Assert.ThatWideString(
	actual := caughtMessage,
	message := "Parse an array root"
).ToBe(expected := "Invalid JSON configuration: not an object");

_Doc := '12345';

caughtMessage := TOF_Core.WideStrings.Empty;

__TRY
	root := _Reader.Parse(document := _Doc);
__CATCH(exceptionCode)
	caughtMessage := getInvalidDocumentMessage(
		exceptionCode := exceptionCode,
		catchPointPOUName := __POUNAME(),
		catchPointPosition := __POSITION()
	);
__ENDTRY

Assert.ThatWideString(
	actual := caughtMessage,
	message := "Parse a scalar root"
).ToBe(expected := "Invalid JSON configuration: not an object");
END_METHOD

(*!
<summary>Verifies successful document open with an object root.</summary>
*)
METHOD PRIVATE testOpenObjectRoot
VAR
	root : TOF_Core.CONFIGURATION_NODE;
END_VAR
_Doc := '{"key": 123}';
root := _Reader.Parse(document := _Doc);

Assert.ThatBool(actual := _Reader.IsPresent(node := root)).IsTrue();
END_METHOD

(*!
<summary>Verifies destination validation, shape checking, type mismatch and capacity errors in ReadValue.</summary>
*)
METHOD PRIVATE testReadValueValidationAndErrors
VAR
	root : TOF_Core.CONFIGURATION_NODE;
	numNode : TOF_Core.CONFIGURATION_NODE;
	strNode : TOF_Core.CONFIGURATION_NODE;
	nullNode : TOF_Core.CONFIGURATION_NODE;
	arrNode : TOF_Core.CONFIGURATION_NODE;
	objNode : TOF_Core.CONFIGURATION_NODE;
	emptyNode : TOF_Core.CONFIGURATION_NODE;
	dstDint : DINT;
	dstStr : STRING(80);
	tinyStr : STRING(2);
END_VAR
_Doc := '{"num": 42, "str": "hello world", "nullVal": null, "arr": [1], "obj": {}}';
root := _Reader.Parse(document := _Doc);
numNode := _Reader.GetField(node := root, name := 'num');
strNode := _Reader.GetField(node := root, name := 'str');
nullNode := _Reader.GetField(node := root, name := 'nullVal');
arrNode := _Reader.GetField(node := root, name := 'arr');
objNode := _Reader.GetField(node := root, name := 'obj');

expectReadValueFailure(
	node := numNode,
	valueType := TOF_Core.CONFIGURATION_VALUE_TYPE.TYPE_DINT,
	data := 0,
	size := 4,
	message := "ReadValue with a null destination",
	expected := "Invalid JSON configuration: type/size mismatch"
);

expectReadValueFailure(
	node := numNode,
	valueType := TOF_Core.CONFIGURATION_VALUE_TYPE.TYPE_DINT,
	data := ADR(dstDint),
	size := 0,
	message := "ReadValue with zero destination size",
	expected := "Invalid JSON configuration: type/size mismatch"
);

expectReadValueFailure(
	node := emptyNode,
	valueType := TOF_Core.CONFIGURATION_VALUE_TYPE.TYPE_DINT,
	data := ADR(dstDint),
	size := 4,
	message := "ReadValue with an absent node",
	expected := "Invalid JSON configuration: missing field"
);

expectReadValueFailure(
	node := nullNode,
	valueType := TOF_Core.CONFIGURATION_VALUE_TYPE.TYPE_DINT,
	data := ADR(dstDint),
	size := 4,
	message := "ReadValue on a null value",
	expected := "Invalid JSON configuration: type/size mismatch"
);

expectReadValueFailure(
	node := arrNode,
	valueType := TOF_Core.CONFIGURATION_VALUE_TYPE.TYPE_DINT,
	data := ADR(dstDint),
	size := 4,
	message := "ReadValue on an array",
	expected := "Invalid JSON configuration: type/size mismatch"
);

expectReadValueFailure(
	node := objNode,
	valueType := TOF_Core.CONFIGURATION_VALUE_TYPE.TYPE_DINT,
	data := ADR(dstDint),
	size := 4,
	message := "ReadValue on an object",
	expected := "Invalid JSON configuration: type/size mismatch"
);

expectReadValueFailure(
	node := numNode,
	valueType := TOF_Core.CONFIGURATION_VALUE_TYPE.TYPE_DINT,
	data := ADR(dstDint),
	size := 3,
	message := "ReadValue with the wrong DINT size",
	expected := "Invalid JSON configuration: type/size mismatch"
);

// SA0175: ReadValue targets a raw string buffer; no character indexing is performed.
{analysis -175}
expectReadValueFailure(
	node := numNode,
	valueType := TOF_Core.CONFIGURATION_VALUE_TYPE.TYPE_STRING,
	data := ADR(dstStr),
	size := SIZEOF(dstStr),
	message := "ReadValue into STRING from a number",
	expected := "Invalid JSON configuration: type/size mismatch"
);

expectReadValueFailure(
	node := strNode,
	valueType := TOF_Core.CONFIGURATION_VALUE_TYPE.TYPE_STRING,
	data := ADR(tinyStr),
	size := SIZEOF(tinyStr),
	message := "ReadValue into an undersized string buffer",
	expected := "Invalid JSON configuration: CopyString failed for STRING(2) (3 destination bytes)"
);
{analysis +175}
END_METHOD

(*!
<summary>Checks empty and ASCII WSTRING values, exact-fit Unicode decoding, and distinguishes a null escape from literal backslash text.</summary>
*)
METHOD PRIVATE testReadWideString
VAR
	root : TOF_Core.CONFIGURATION_NODE;
	unicodeNode : TOF_Core.CONFIGURATION_NODE;
	wideText : WSTRING(2);
	shortText : WSTRING(1) := "X";
	literalText : WSTRING(6);
END_VAR
_Doc := '{"name":"AB","emptyName":"","unicode":"\u00e9\u0416","withNull":"A\u0000B","literal":"\\u0000"}';
root := _Reader.Parse(document := _Doc);

_Reader.ReadValue(
	node := _Reader.GetField(node := root, name := 'name'),
	valueType := TOF_Core.CONFIGURATION_VALUE_TYPE.TYPE_WSTRING,
	data := ADR(wideText),
	size := SIZEOF(wideText)
);
Assert.ThatWideString(actual := wideText, message := "Read an ASCII name").ToBe(expected := "AB");

_Reader.ReadValue(
	node := _Reader.GetField(node := root, name := 'emptyName'),
	valueType := TOF_Core.CONFIGURATION_VALUE_TYPE.TYPE_WSTRING,
	data := ADR(wideText),
	size := SIZEOF(wideText)
);
Assert.ThatWideString(actual := wideText, message := "An empty name clears the previous value").ToBe(expected := "");

unicodeNode := _Reader.GetField(node := root, name := 'unicode');

_Reader.ReadValue(
	node := unicodeNode,
	valueType := TOF_Core.CONFIGURATION_VALUE_TYPE.TYPE_WSTRING,
	data := ADR(wideText),
	size := SIZEOF(wideText)
);
Assert.ThatWideString(actual := wideText, message := "Decode two Unicode characters into two wide slots").ToBe(
	expected := "$00E9$0416"
);

expectReadValueFailure(
	node := unicodeNode,
	valueType := TOF_Core.CONFIGURATION_VALUE_TYPE.TYPE_WSTRING,
	data := ADR(shortText),
	size := SIZEOF(shortText),
	message := "Reject a WSTRING destination with room for only one character",
	expected := "Invalid JSON configuration: WSTRING needs 2 characters, capacity 1"
);
Assert.ThatWideString(actual := shortText, message := "Capacity failure must precede conversion").ToBe(expected := "X");

_Reader.ReadValue(
	node := _Reader.GetField(node := root, name := 'literal'),
	valueType := TOF_Core.CONFIGURATION_VALUE_TYPE.TYPE_WSTRING,
	data := ADR(literalText),
	size := SIZEOF(literalText)
);
Assert.ThatWideString(actual := literalText, message := "Preserve a literal backslash").ToBe(expected := "\u0000");

expectReadValueFailure(
	node := _Reader.GetField(node := root, name := 'withNull'),
	valueType := TOF_Core.CONFIGURATION_VALUE_TYPE.TYPE_WSTRING,
	data := ADR(wideText),
	size := SIZEOF(wideText),
	message := "Reject embedded null in JSON string",
	expected := "Invalid JSON configuration: parse failure"
);
END_METHOD

(*!
<summary>Verifies that a new document can be parsed and read using newly obtained cursors.</summary>
*)
METHOD PRIVATE testReparseReadsNewDocument
VAR
	root1 : TOF_Core.CONFIGURATION_NODE;
	root2 : TOF_Core.CONFIGURATION_NODE;
	nodeVal : TOF_Core.CONFIGURATION_NODE;
	val : DINT;
END_VAR
_Doc := '{"id": 1}';
root1 := _Reader.Parse(document := _Doc);
nodeVal := _Reader.GetField(node := root1, name := 'id');
_Reader.ReadValue(
	node := nodeVal,
	valueType := TOF_Core.CONFIGURATION_VALUE_TYPE.TYPE_DINT,
	data := ADR(val),
	size := SIZEOF(val)
);
Assert.ThatDInt(actual := val).ToBe(expected := 1);

_Doc := '{"id": 2}';
root2 := _Reader.Parse(document := _Doc);
nodeVal := _Reader.GetField(node := root2, name := 'id');
_Reader.ReadValue(
	node := nodeVal,
	valueType := TOF_Core.CONFIGURATION_VALUE_TYPE.TYPE_DINT,
	data := ADR(val),
	size := SIZEOF(val)
);
Assert.ThatDInt(actual := val).ToBe(expected := 2);
END_METHOD

(*!
<summary>Verifies that FindField returns an empty node for absent members and non-object parents.</summary>
*)
METHOD PRIVATE testFindOptionalField
VAR
	root : TOF_Core.CONFIGURATION_NODE;
	fieldNode : TOF_Core.CONFIGURATION_NODE;
	missingNode : TOF_Core.CONFIGURATION_NODE;
	emptyParent : TOF_Core.CONFIGURATION_NODE;
	fieldOnEmpty : TOF_Core.CONFIGURATION_NODE;
	fieldOnScalar : TOF_Core.CONFIGURATION_NODE;
END_VAR
_Doc := '{"present": 10}';
root := _Reader.Parse(document := _Doc);

fieldNode := _Reader.FindField(node := root, name := 'present');
Assert.ThatBool(actual := _Reader.IsPresent(node := fieldNode)).IsTrue();

missingNode := _Reader.FindField(node := root, name := 'absent');
Assert.ThatBool(actual := _Reader.IsPresent(node := missingNode)).IsFalse();

fieldOnEmpty := _Reader.FindField(node := emptyParent, name := 'any');
Assert.ThatBool(actual := _Reader.IsPresent(node := fieldOnEmpty)).IsFalse();

fieldOnScalar := _Reader.FindField(node := fieldNode, name := 'any');
Assert.ThatBool(
	actual := _Reader.IsPresent(node := fieldOnScalar),
	message := "FindField on a scalar must return an empty node"
).IsFalse();
END_METHOD

(*!
<summary>Invokes ReadValue with one invalid input and compares the resulting reader diagnostic.</summary>
<description>A valid return or a different exception fails the named scenario.</description>
*)
METHOD PRIVATE expectReadValueFailure
VAR_INPUT
	node : TOF_Core.CONFIGURATION_NODE;
	valueType : TOF_Core.CONFIGURATION_VALUE_TYPE;
	data : PVOID;
	size : UDINT;
	message : WSTRING(255);
	expected : WSTRING(255);
END_VAR
VAR
	caughtMessage : WSTRING(255);
	exceptionCode : __SYSTEM.ExceptionCode;
END_VAR
__TRY
	_Reader.ReadValue(node := node, valueType := valueType, data := data, size := size);
__CATCH(exceptionCode)
	caughtMessage := getInvalidDocumentMessage(
		exceptionCode := exceptionCode,
		catchPointPOUName := __POUNAME(),
		catchPointPosition := __POSITION()
	);
__ENDTRY

Assert.ThatWideString(actual := caughtMessage, message := message).ToBe(expected := expected);
END_METHOD

(*!
<summary>Copies the structured invalid-argument diagnostic from the active catch.</summary>
<description>Unexpected payloads yield a diagnostic that cannot match a valid reader error.</description>
*)
METHOD PRIVATE getInvalidDocumentMessage : WSTRING(255)
VAR_INPUT
	exceptionCode : __SYSTEM.ExceptionCode;
	catchPointPOUName : STRING;
	catchPointPosition : STRING;
END_VAR
VAR
	exception : TOF_Core.IException;
	generalException : TOF_Core.IGeneralException;
END_VAR
exception := TOF_Core.ExceptionManager.GetLastException(
	exceptionCode := exceptionCode,
	catchPointNamespaceName := NamespaceName,
	catchPointPOUName := catchPointPOUName,
	catchPointPosition := catchPointPosition
);

IF exception <> 0 AND_THEN __QUERYINTERFACE(exception, generalException) THEN
	IF generalException.ErrorCode = _InvalidArgumentCode THEN
		getInvalidDocumentMessage := generalException.SourceMessage;
		RETURN;
	END_IF
END_IF

IF exception = 0 THEN
	getInvalidDocumentMessage := "No exception payload";
ELSE
	getInvalidDocumentMessage := TOF_Core.WideStrings.ConcatFit255("Unexpected exception: ", exception.GetMessage());
END_IF
END_METHOD

(*!
<summary>Verifies that a context-free object deserializes successfully with null deserialization context.</summary>
*)
METHOD PRIVATE testDeserializeContextFreeObject
VAR
	root : TOF_Core.CONFIGURATION_NODE;
END_VAR
_Mock.Reset();
_Doc := '{"intField":123,"stringField":"test context-free"}';
root := _Reader.Parse(document := _Doc);
_Mock.Deserialize(reader := _Reader, node := root, context := 0);

Assert.ThatUDInt(actual := _Mock.DeserializeCount).ToBe(expected := 1);
Assert.ThatDInt(actual := _Mock.IntField).ToBe(expected := 123);
Assert.ThatString(actual := _Mock.StringField).ToBe(expected := 'test context-free');
END_METHOD

END_FUNCTION_BLOCK

// ---- Tests/JSON/JsonConfigurationRoundTripTest.TcPOU
(*
SPDX-FileCopyrightText: © 2026 Oleksandr Tiutyk <trofimich@gmail.com>
SPDX-License-Identifier: MIT
License: https://opensource.org/license/mit
*)

(*!
<summary>Exercises full configuration round-trip for all 25 CONFIGURATION_VALUE_TYPE values.</summary>
<description>
Verifies serialization and deserialization symmetry across boundary values of all integer, bitstring,
floating-point, string, wide string and date/time types, as well as nested objects, lists, and empty strings.
</description>
*)

{attribute 'no_assign'}
{attribute 'no_explicit_call' := 'do not call this function block directly'}
FUNCTION_BLOCK JsonConfigurationRoundTripTest EXTENDS TOF_Testing.SingleCycleTest
VAR_STAT
	{attribute 'hide'}
	_ClassName : STRING := __POUNAME();
END_VAR
VAR
	{attribute 'hide'}
	{attribute 'init_namespace'}
	_NamespaceName : STRING;
END_VAR
VAR
	_Writer : TOF_JSON.JsonConfigurationWriter;
	_Reader : TOF_JSON.JsonConfigurationReader;
	_Dom : Tc3_JsonXml.FB_JsonDomParser;
	_ReferenceConverter : Tc3_JsonXml.FB_JsonReadWriteDataType;
	_Doc : TOF_Core.JSON_DOCUMENT;
END_VAR

(*!
<summary>Borrows the concrete class name for the lifetime of this instance.</summary>
*)
{attribute 'monitoring' := 'call'}
PROPERTY ClassName : REFERENCE TO STRING
GET
ClassName REF= _ClassName;
END_GET
END_PROPERTY

(*!
<summary>Exercises JSON round trips for elementary values and nested objects and arrays.</summary>
*)
METHOD PROTECTED ExecuteTest
testIntegerTypesRoundTrip();
testBitStringTypesRoundTrip();
testFloatTypesRoundTrip();
testStringsRoundTrip();
testWideStringsRoundTrip();
testDateTimeTypesRoundTrip();
testStructuralRoundTrip();
END_METHOD

(*!
<summary>Borrows the compiler-initialized namespace for the lifetime of this instance.</summary>
*)
{attribute 'monitoring' := 'call'}
PROPERTY NamespaceName : REFERENCE TO STRING
GET
NamespaceName REF= CurrentNamespace.Name;
END_GET
END_PROPERTY

(*!
<summary>Reports the complete concrete instance size in bytes.</summary>
*)
{attribute 'monitoring' := 'call'}
PROPERTY SelfSize : ULINT
GET
SelfSize := XSIZEOF(THIS^);
END_GET
END_PROPERTY

(*!
<summary>Verifies round-trip serialization of BOOL, BYTE, WORD, DWORD and LWORD bitstring types.</summary>
*)
METHOD PRIVATE testBitStringTypesRoundTrip
VAR
	root : TOF_Core.CONFIGURATION_NODE;
	boolTrue : BOOL := TRUE;
	boolFalse : BOOL := FALSE;
	byteVal : BYTE := 16#AB;
	wordVal : WORD := 16#ABCD;
	dwordVal : DWORD := 16#12345678;
	lwordVal : LWORD := 16#0123456789ABCDEF;
	boolDst : BOOL;
	byteDst : BYTE;
	wordDst : WORD;
	dwordDst : DWORD;
	lwordDst : LWORD;
END_VAR
_Writer.BeginDocument();
_Writer.WriteValue(
	name := 'bTrue',
	valueType := TOF_Core.CONFIGURATION_VALUE_TYPE.TYPE_BOOL,
	data := ADR(boolTrue),
	size := SIZEOF(boolTrue)
);
_Writer.WriteValue(
	name := 'bFalse',
	valueType := TOF_Core.CONFIGURATION_VALUE_TYPE.TYPE_BOOL,
	data := ADR(boolFalse),
	size := SIZEOF(boolFalse)
);
_Writer.WriteValue(
	name := 'byteV',
	valueType := TOF_Core.CONFIGURATION_VALUE_TYPE.TYPE_BYTE,
	data := ADR(byteVal),
	size := SIZEOF(byteVal)
);
_Writer.WriteValue(
	name := 'wordV',
	valueType := TOF_Core.CONFIGURATION_VALUE_TYPE.TYPE_WORD,
	data := ADR(wordVal),
	size := SIZEOF(wordVal)
);
_Writer.WriteValue(
	name := 'dwordV',
	valueType := TOF_Core.CONFIGURATION_VALUE_TYPE.TYPE_DWORD,
	data := ADR(dwordVal),
	size := SIZEOF(dwordVal)
);
_Writer.WriteValue(
	name := 'lwordV',
	valueType := TOF_Core.CONFIGURATION_VALUE_TYPE.TYPE_LWORD,
	data := ADR(lwordVal),
	size := SIZEOF(lwordVal)
);
_Writer.EndDocument(document := _Doc);

root := _Reader.Parse(document := _Doc);

_Reader.ReadValue(
	node := _Reader.GetField(node := root, name := 'bTrue'),
	valueType := TOF_Core.CONFIGURATION_VALUE_TYPE.TYPE_BOOL,
	data := ADR(boolDst),
	size := SIZEOF(boolDst)
);
Assert.ThatBool(actual := boolDst).IsTrue();

_Reader.ReadValue(
	node := _Reader.GetField(node := root, name := 'bFalse'),
	valueType := TOF_Core.CONFIGURATION_VALUE_TYPE.TYPE_BOOL,
	data := ADR(boolDst),
	size := SIZEOF(boolDst)
);
Assert.ThatBool(actual := boolDst).IsFalse();

_Reader.ReadValue(
	node := _Reader.GetField(node := root, name := 'byteV'),
	valueType := TOF_Core.CONFIGURATION_VALUE_TYPE.TYPE_BYTE,
	data := ADR(byteDst),
	size := SIZEOF(byteDst)
);
Assert.ThatByte(actual := byteDst).ToBe(expected := 16#AB);

_Reader.ReadValue(
	node := _Reader.GetField(node := root, name := 'wordV'),
	valueType := TOF_Core.CONFIGURATION_VALUE_TYPE.TYPE_WORD,
	data := ADR(wordDst),
	size := SIZEOF(wordDst)
);
Assert.ThatWord(actual := wordDst).ToBe(expected := 16#ABCD);

_Reader.ReadValue(
	node := _Reader.GetField(node := root, name := 'dwordV'),
	valueType := TOF_Core.CONFIGURATION_VALUE_TYPE.TYPE_DWORD,
	data := ADR(dwordDst),
	size := SIZEOF(dwordDst)
);
Assert.ThatDWord(actual := dwordDst).ToBe(expected := 16#12345678);

_Reader.ReadValue(
	node := _Reader.GetField(node := root, name := 'lwordV'),
	valueType := TOF_Core.CONFIGURATION_VALUE_TYPE.TYPE_LWORD,
	data := ADR(lwordDst),
	size := SIZEOF(lwordDst)
);
Assert.ThatLWord(actual := lwordDst).ToBe(expected := 16#0123456789ABCDEF);
END_METHOD

(*!
<summary>Verifies round-trip serialization of eight time types and compares LTIME with direct native serialization.</summary>
*)
METHOD PRIVATE testDateTimeTypesRoundTrip
VAR
	root : TOF_Core.CONFIGURATION_NODE;
	domRoot : Tc3_JsonXml.SJsonValue;
	serializedTime : Tc3_JsonXml.SJsonValue;
	referenceJson : STRING(255);
	referenceSize : UDINT;
	actualJson : STRING(255);
	timeVal : TIME := T#49D17H2M47S295MS;
	ltimeVal : LTIME := LTIME#100D12H30M15S;
	dateVal : DATE := D#2026-11-09;
	ldateVal : LDATE := LDATE#2026-11-09;
	todVal : TOD := TOD#14:30:15.500;
	ltodVal : LTOD := LTOD#14:30:15.123456789;
	dtVal : DT := DT#2026-11-09-14:30:15;
	ldtVal : LDT := LDT#2026-11-09-14:30:15.123456789;
	timeDst : TIME;
	ltimeDst : LTIME;
	dateDst : DATE;
	ldateDst : LDATE;
	todDst : TOD;
	ltodDst : LTOD;
	dtDst : DT;
	ldtDst : LDT;
END_VAR
_Writer.BeginDocument();
_Writer.WriteValue(
	name := 'timeV',
	valueType := TOF_Core.CONFIGURATION_VALUE_TYPE.TYPE_TIME,
	data := ADR(timeVal),
	size := SIZEOF(timeVal)
);
_Writer.WriteValue(
	name := 'ltimeV',
	valueType := TOF_Core.CONFIGURATION_VALUE_TYPE.TYPE_LTIME,
	data := ADR(ltimeVal),
	size := SIZEOF(ltimeVal)
);
_Writer.WriteValue(
	name := 'dateV',
	valueType := TOF_Core.CONFIGURATION_VALUE_TYPE.TYPE_DATE,
	data := ADR(dateVal),
	size := SIZEOF(dateVal)
);
_Writer.WriteValue(
	name := 'ldateV',
	valueType := TOF_Core.CONFIGURATION_VALUE_TYPE.TYPE_LDATE,
	data := ADR(ldateVal),
	size := SIZEOF(ldateVal)
);
_Writer.WriteValue(
	name := 'todV',
	valueType := TOF_Core.CONFIGURATION_VALUE_TYPE.TYPE_TOD,
	data := ADR(todVal),
	size := SIZEOF(todVal)
);
_Writer.WriteValue(
	name := 'ltodV',
	valueType := TOF_Core.CONFIGURATION_VALUE_TYPE.TYPE_LTOD,
	data := ADR(ltodVal),
	size := SIZEOF(ltodVal)
);
_Writer.WriteValue(
	name := 'dtV',
	valueType := TOF_Core.CONFIGURATION_VALUE_TYPE.TYPE_DT,
	data := ADR(dtVal),
	size := SIZEOF(dtVal)
);
_Writer.WriteValue(
	name := 'ldtV',
	valueType := TOF_Core.CONFIGURATION_VALUE_TYPE.TYPE_LDT,
	data := ADR(ldtVal),
	size := SIZEOF(ldtVal)
);
_Writer.EndDocument(document := _Doc);

referenceSize := SIZEOF(referenceJson);

// SA0175: GetJsonFromSymbol writes to the string buffer using its size in bytes.
{analysis -175}
IF NOT _ReferenceConverter.GetJsonFromSymbol(
	sDatatype := 'LTIME',
	nData := SIZEOF(ltimeVal),
	pData := ADR(ltimeVal),
	nJson := referenceSize,
	pJson := ADR(referenceJson)
) THEN
	RecordFailure(message := "Native LTIME reference serialization failed");
	RETURN;
END_IF
{analysis +175}

domRoot := _Dom.ParseDocument(sJson := _Doc);

IF domRoot = 0 OR_ELSE NOT _Dom.IsObject(v := domRoot) THEN
	RecordFailure(message := "Serialized temporal values must form a JSON object");
	RETURN;
END_IF

serializedTime := _Dom.FindMember(v := domRoot, member := 'ltimeV');

IF serializedTime = 0 THEN
	RecordFailure(message := "The serialized document must contain ltimeV");
	RETURN;
END_IF

IF _Dom.CopyJson(v := serializedTime, pDoc := actualJson, nDoc := SIZEOF(actualJson)) = 0 THEN
	RecordFailure(message := "Could not read the serialized ltimeV JSON value");
	RETURN;
END_IF

Assert.ThatString(actual := actualJson, message := "LTIME JSON must match its native representation").ToBe(
	expected := referenceJson
);

root := _Reader.Parse(document := _Doc);

_Reader.ReadValue(
	node := _Reader.GetField(node := root, name := 'timeV'),
	valueType := TOF_Core.CONFIGURATION_VALUE_TYPE.TYPE_TIME,
	data := ADR(timeDst),
	size := SIZEOF(timeDst)
);
Assert.ThatTime(actual := timeDst).ToBe(expected := timeVal);

_Reader.ReadValue(
	node := _Reader.GetField(node := root, name := 'ltimeV'),
	valueType := TOF_Core.CONFIGURATION_VALUE_TYPE.TYPE_LTIME,
	data := ADR(ltimeDst),
	size := SIZEOF(ltimeDst)
);
Assert.ThatLongTime(actual := ltimeDst).ToBe(expected := ltimeVal);

_Reader.ReadValue(
	node := _Reader.GetField(node := root, name := 'dateV'),
	valueType := TOF_Core.CONFIGURATION_VALUE_TYPE.TYPE_DATE,
	data := ADR(dateDst),
	size := SIZEOF(dateDst)
);
Assert.ThatDate(actual := dateDst).ToBe(expected := dateVal);

_Reader.ReadValue(
	node := _Reader.GetField(node := root, name := 'ldateV'),
	valueType := TOF_Core.CONFIGURATION_VALUE_TYPE.TYPE_LDATE,
	data := ADR(ldateDst),
	size := SIZEOF(ldateDst)
);
Assert.ThatLongDate(actual := ldateDst).ToBe(expected := ldateVal);

_Reader.ReadValue(
	node := _Reader.GetField(node := root, name := 'todV'),
	valueType := TOF_Core.CONFIGURATION_VALUE_TYPE.TYPE_TOD,
	data := ADR(todDst),
	size := SIZEOF(todDst)
);
Assert.ThatTimeOfDay(actual := todDst).ToBe(expected := todVal);

_Reader.ReadValue(
	node := _Reader.GetField(node := root, name := 'ltodV'),
	valueType := TOF_Core.CONFIGURATION_VALUE_TYPE.TYPE_LTOD,
	data := ADR(ltodDst),
	size := SIZEOF(ltodDst)
);
Assert.ThatLongTimeOfDay(actual := ltodDst).ToBe(expected := ltodVal);

_Reader.ReadValue(
	node := _Reader.GetField(node := root, name := 'dtV'),
	valueType := TOF_Core.CONFIGURATION_VALUE_TYPE.TYPE_DT,
	data := ADR(dtDst),
	size := SIZEOF(dtDst)
);
Assert.ThatDateTime(actual := dtDst).ToBe(expected := dtVal);

_Reader.ReadValue(
	node := _Reader.GetField(node := root, name := 'ldtV'),
	valueType := TOF_Core.CONFIGURATION_VALUE_TYPE.TYPE_LDT,
	data := ADR(ldtDst),
	size := SIZEOF(ldtDst)
);
Assert.ThatLongDateTime(actual := ldtDst).ToBe(expected := ldtVal);
END_METHOD

(*!
<summary>Verifies round-trip serialization of REAL and LREAL floating point types within tolerance.</summary>
*)
METHOD PRIVATE testFloatTypesRoundTrip
VAR
	root : TOF_Core.CONFIGURATION_NODE;
	realPos : REAL := 123.456;
	realNeg : REAL := -123.456;
	lrealPos : LREAL := 987654.3210123;
	lrealNeg : LREAL := -987654.3210123;
	realDst : REAL;
	lrealDst : LREAL;
END_VAR
_Writer.BeginDocument();
_Writer.WriteValue(
	name := 'rPos',
	valueType := TOF_Core.CONFIGURATION_VALUE_TYPE.TYPE_REAL,
	data := ADR(realPos),
	size := SIZEOF(realPos)
);
_Writer.WriteValue(
	name := 'rNeg',
	valueType := TOF_Core.CONFIGURATION_VALUE_TYPE.TYPE_REAL,
	data := ADR(realNeg),
	size := SIZEOF(realNeg)
);
_Writer.WriteValue(
	name := 'lrPos',
	valueType := TOF_Core.CONFIGURATION_VALUE_TYPE.TYPE_LREAL,
	data := ADR(lrealPos),
	size := SIZEOF(lrealPos)
);
_Writer.WriteValue(
	name := 'lrNeg',
	valueType := TOF_Core.CONFIGURATION_VALUE_TYPE.TYPE_LREAL,
	data := ADR(lrealNeg),
	size := SIZEOF(lrealNeg)
);
_Writer.EndDocument(document := _Doc);

root := _Reader.Parse(document := _Doc);

_Reader.ReadValue(
	node := _Reader.GetField(node := root, name := 'rPos'),
	valueType := TOF_Core.CONFIGURATION_VALUE_TYPE.TYPE_REAL,
	data := ADR(realDst),
	size := SIZEOF(realDst)
);
Assert.ThatReal(actual := realDst).ToBe(expected := 123.456, tolerance := 0.01);

_Reader.ReadValue(
	node := _Reader.GetField(node := root, name := 'rNeg'),
	valueType := TOF_Core.CONFIGURATION_VALUE_TYPE.TYPE_REAL,
	data := ADR(realDst),
	size := SIZEOF(realDst)
);
Assert.ThatReal(actual := realDst).ToBe(expected := -123.456, tolerance := 0.01);

_Reader.ReadValue(
	node := _Reader.GetField(node := root, name := 'lrPos'),
	valueType := TOF_Core.CONFIGURATION_VALUE_TYPE.TYPE_LREAL,
	data := ADR(lrealDst),
	size := SIZEOF(lrealDst)
);
Assert.ThatLongReal(actual := lrealDst).ToBe(expected := 987654.3210123, tolerance := 0.0001);

_Reader.ReadValue(
	node := _Reader.GetField(node := root, name := 'lrNeg'),
	valueType := TOF_Core.CONFIGURATION_VALUE_TYPE.TYPE_LREAL,
	data := ADR(lrealDst),
	size := SIZEOF(lrealDst)
);
Assert.ThatLongReal(actual := lrealDst).ToBe(expected := -987654.3210123, tolerance := 0.0001);
END_METHOD

(*!
<summary>Verifies round-trip and exact JSON numeric values at representative signed and unsigned integer boundaries.</summary>
*)
METHOD PRIVATE testIntegerTypesRoundTrip
VAR
	root : TOF_Core.CONFIGURATION_NODE;
	domRoot : Tc3_JsonXml.SJsonValue;
	number : Tc3_JsonXml.SJsonValue;
	sintMin : SINT := -128;
	sintMax : SINT := 127;
	usintMax : USINT := 255;
	intMin : INT := -32768;
	intMax : INT := 32767;
	uintMax : UINT := 65535;
	dintMin : DINT := -2147483648;
	dintMax : DINT := 2147483647;
	udintMax : UDINT := 4294967295;
	lintVal : LINT := -9223372036854775807;
	ulintVal : ULINT := 18446744073709551615;
	sintDst : SINT;
	usintDst : USINT;
	intDst : INT;
	uintDst : UINT;
	dintDst : DINT;
	udintDst : UDINT;
	lintDst : LINT;
	ulintDst : ULINT;
END_VAR
_Writer.BeginDocument();
_Writer.WriteValue(
	name := 'sintMin',
	valueType := TOF_Core.CONFIGURATION_VALUE_TYPE.TYPE_SINT,
	data := ADR(sintMin),
	size := SIZEOF(sintMin)
);
_Writer.WriteValue(
	name := 'sintMax',
	valueType := TOF_Core.CONFIGURATION_VALUE_TYPE.TYPE_SINT,
	data := ADR(sintMax),
	size := SIZEOF(sintMax)
);
_Writer.WriteValue(
	name := 'usintMax',
	valueType := TOF_Core.CONFIGURATION_VALUE_TYPE.TYPE_USINT,
	data := ADR(usintMax),
	size := SIZEOF(usintMax)
);
_Writer.WriteValue(
	name := 'intMin',
	valueType := TOF_Core.CONFIGURATION_VALUE_TYPE.TYPE_INT,
	data := ADR(intMin),
	size := SIZEOF(intMin)
);
_Writer.WriteValue(
	name := 'intMax',
	valueType := TOF_Core.CONFIGURATION_VALUE_TYPE.TYPE_INT,
	data := ADR(intMax),
	size := SIZEOF(intMax)
);
_Writer.WriteValue(
	name := 'uintMax',
	valueType := TOF_Core.CONFIGURATION_VALUE_TYPE.TYPE_UINT,
	data := ADR(uintMax),
	size := SIZEOF(uintMax)
);
_Writer.WriteValue(
	name := 'dintMin',
	valueType := TOF_Core.CONFIGURATION_VALUE_TYPE.TYPE_DINT,
	data := ADR(dintMin),
	size := SIZEOF(dintMin)
);
_Writer.WriteValue(
	name := 'dintMax',
	valueType := TOF_Core.CONFIGURATION_VALUE_TYPE.TYPE_DINT,
	data := ADR(dintMax),
	size := SIZEOF(dintMax)
);
_Writer.WriteValue(
	name := 'udintMax',
	valueType := TOF_Core.CONFIGURATION_VALUE_TYPE.TYPE_UDINT,
	data := ADR(udintMax),
	size := SIZEOF(udintMax)
);
_Writer.WriteValue(
	name := 'lintV',
	valueType := TOF_Core.CONFIGURATION_VALUE_TYPE.TYPE_LINT,
	data := ADR(lintVal),
	size := SIZEOF(lintVal)
);
_Writer.WriteValue(
	name := 'ulintV',
	valueType := TOF_Core.CONFIGURATION_VALUE_TYPE.TYPE_ULINT,
	data := ADR(ulintVal),
	size := SIZEOF(ulintVal)
);
_Writer.EndDocument(document := _Doc);

domRoot := _Dom.ParseDocument(sJson := _Doc);

IF domRoot = 0 OR_ELSE NOT _Dom.IsObject(v := domRoot) THEN
	RecordFailure(message := "Serialized integer values must form a JSON object");
	RETURN;
END_IF

number := _Dom.FindMember(v := domRoot, member := 'lintV');

IF number = 0 OR_ELSE NOT _Dom.IsInt64(v := number) THEN
	RecordFailure(message := "lintV must remain a signed 64-bit JSON integer");
	RETURN;
END_IF

Assert.ThatLInt(actual := _Dom.GetInt64(v := number), message := "Signed 64-bit JSON value").ToBe(
	expected := lintVal
);

number := _Dom.FindMember(v := domRoot, member := 'ulintV');

IF number = 0 OR_ELSE NOT _Dom.IsUint64(v := number) THEN
	RecordFailure(message := "ulintV must remain an unsigned 64-bit JSON integer");
	RETURN;
END_IF

Assert.ThatULInt(actual := _Dom.GetUint64(v := number), message := "Unsigned 64-bit JSON value").ToBe(
	expected := ulintVal
);

root := _Reader.Parse(document := _Doc);

_Reader.ReadValue(
	node := _Reader.GetField(node := root, name := 'sintMin'),
	valueType := TOF_Core.CONFIGURATION_VALUE_TYPE.TYPE_SINT,
	data := ADR(sintDst),
	size := SIZEOF(sintDst)
);
Assert.ThatSInt(actual := sintDst).ToBe(expected := -128);

_Reader.ReadValue(
	node := _Reader.GetField(node := root, name := 'sintMax'),
	valueType := TOF_Core.CONFIGURATION_VALUE_TYPE.TYPE_SINT,
	data := ADR(sintDst),
	size := SIZEOF(sintDst)
);
Assert.ThatSInt(actual := sintDst).ToBe(expected := 127);

_Reader.ReadValue(
	node := _Reader.GetField(node := root, name := 'usintMax'),
	valueType := TOF_Core.CONFIGURATION_VALUE_TYPE.TYPE_USINT,
	data := ADR(usintDst),
	size := SIZEOF(usintDst)
);
Assert.ThatUSInt(actual := usintDst).ToBe(expected := 255);

_Reader.ReadValue(
	node := _Reader.GetField(node := root, name := 'intMin'),
	valueType := TOF_Core.CONFIGURATION_VALUE_TYPE.TYPE_INT,
	data := ADR(intDst),
	size := SIZEOF(intDst)
);
Assert.ThatInt(actual := intDst).ToBe(expected := -32768);

_Reader.ReadValue(
	node := _Reader.GetField(node := root, name := 'intMax'),
	valueType := TOF_Core.CONFIGURATION_VALUE_TYPE.TYPE_INT,
	data := ADR(intDst),
	size := SIZEOF(intDst)
);
Assert.ThatInt(actual := intDst).ToBe(expected := 32767);

_Reader.ReadValue(
	node := _Reader.GetField(node := root, name := 'uintMax'),
	valueType := TOF_Core.CONFIGURATION_VALUE_TYPE.TYPE_UINT,
	data := ADR(uintDst),
	size := SIZEOF(uintDst)
);
Assert.ThatUInt(actual := uintDst).ToBe(expected := 65535);

_Reader.ReadValue(
	node := _Reader.GetField(node := root, name := 'dintMin'),
	valueType := TOF_Core.CONFIGURATION_VALUE_TYPE.TYPE_DINT,
	data := ADR(dintDst),
	size := SIZEOF(dintDst)
);
Assert.ThatDInt(actual := dintDst).ToBe(expected := -2147483648);

_Reader.ReadValue(
	node := _Reader.GetField(node := root, name := 'dintMax'),
	valueType := TOF_Core.CONFIGURATION_VALUE_TYPE.TYPE_DINT,
	data := ADR(dintDst),
	size := SIZEOF(dintDst)
);
Assert.ThatDInt(actual := dintDst).ToBe(expected := 2147483647);

_Reader.ReadValue(
	node := _Reader.GetField(node := root, name := 'udintMax'),
	valueType := TOF_Core.CONFIGURATION_VALUE_TYPE.TYPE_UDINT,
	data := ADR(udintDst),
	size := SIZEOF(udintDst)
);
Assert.ThatUDInt(actual := udintDst).ToBe(expected := 4294967295);

_Reader.ReadValue(
	node := _Reader.GetField(node := root, name := 'lintV'),
	valueType := TOF_Core.CONFIGURATION_VALUE_TYPE.TYPE_LINT,
	data := ADR(lintDst),
	size := SIZEOF(lintDst)
);
Assert.ThatLInt(actual := lintDst).ToBe(expected := lintVal);

_Reader.ReadValue(
	node := _Reader.GetField(node := root, name := 'ulintV'),
	valueType := TOF_Core.CONFIGURATION_VALUE_TYPE.TYPE_ULINT,
	data := ADR(ulintDst),
	size := SIZEOF(ulintDst)
);
Assert.ThatULInt(actual := ulintDst).ToBe(expected := ulintVal);
END_METHOD

(*!
<summary>Verifies empty and escaped strings using a literal JSON fixture and native DOM decoding.</summary>
*)
METHOD PRIVATE testStringsRoundTrip
VAR
	root : TOF_Core.CONFIGURATION_NODE;
	domRoot : Tc3_JsonXml.SJsonValue;
	escapedValue : Tc3_JsonXml.SJsonValue;
	emptySrc : STRING(80) := '';
	regSrc : STRING(80) := 'Hello Structured World';
	escapeSrc : STRING(80) := 'Line1$NLine2$T"Quoted"\';
	strDst : STRING(80) := 'initial';
END_VAR
// SA0175: Raw string buffer binding for JSON round-trip tests; no character indexing.
{analysis -175}
_Writer.BeginDocument();
_Writer.WriteValue(
	name := 'emptyStr',
	valueType := TOF_Core.CONFIGURATION_VALUE_TYPE.TYPE_STRING,
	data := ADR(emptySrc),
	size := SIZEOF(emptySrc)
);
_Writer.WriteValue(
	name := 'regStr',
	valueType := TOF_Core.CONFIGURATION_VALUE_TYPE.TYPE_STRING,
	data := ADR(regSrc),
	size := SIZEOF(regSrc)
);
_Writer.WriteValue(
	name := 'escapeStr',
	valueType := TOF_Core.CONFIGURATION_VALUE_TYPE.TYPE_STRING,
	data := ADR(escapeSrc),
	size := SIZEOF(escapeSrc)
);
_Writer.EndDocument(document := _Doc);

domRoot := _Dom.ParseDocument(sJson := _Doc);

IF domRoot = 0 OR_ELSE NOT _Dom.IsObject(v := domRoot) THEN
	RecordFailure(message := "Serialized STRING values must form a JSON object");
	RETURN;
END_IF

escapedValue := _Dom.FindMember(v := domRoot, member := 'escapeStr');

IF escapedValue = 0 OR_ELSE NOT _Dom.IsString(v := escapedValue) THEN
	RecordFailure(message := "escapeStr must be a JSON string");
	RETURN;
END_IF

Assert.ThatString(actual := _Dom.GetString(v := escapedValue), message := "DOM-decoded escaped value").ToBe(
	expected := 'Line1$NLine2$T"Quoted"\'
);

root := _Reader.Parse(document := _Doc);

_Reader.ReadValue(
	node := _Reader.GetField(node := root, name := 'emptyStr'),
	valueType := TOF_Core.CONFIGURATION_VALUE_TYPE.TYPE_STRING,
	data := ADR(strDst),
	size := SIZEOF(strDst)
);
Assert.ThatString(actual := strDst).ToBe(expected := '');

_Reader.ReadValue(
	node := _Reader.GetField(node := root, name := 'regStr'),
	valueType := TOF_Core.CONFIGURATION_VALUE_TYPE.TYPE_STRING,
	data := ADR(strDst),
	size := SIZEOF(strDst)
);
Assert.ThatString(actual := strDst).ToBe(expected := 'Hello Structured World');

_Reader.ReadValue(
	node := _Reader.GetField(node := root, name := 'escapeStr'),
	valueType := TOF_Core.CONFIGURATION_VALUE_TYPE.TYPE_STRING,
	data := ADR(strDst),
	size := SIZEOF(strDst)
);
Assert.ThatString(actual := strDst).ToBe(expected := 'Line1$NLine2$T"Quoted"\');

// Pure reader test on manual JSON with empty string
_Doc := '{"standaloneEmpty": ""}';
root := _Reader.Parse(document := _Doc);
strDst := 'initial';
_Reader.ReadValue(
	node := _Reader.GetField(node := root, name := 'standaloneEmpty'),
	valueType := TOF_Core.CONFIGURATION_VALUE_TYPE.TYPE_STRING,
	data := ADR(strDst),
	size := SIZEOF(strDst)
);
{analysis +175}
Assert.ThatString(actual := strDst).ToBe(expected := '');
END_METHOD

(*!
<summary>Verifies round-trip for nested configuration objects and ordered lists.</summary>
*)
METHOD PRIVATE testStructuralRoundTrip
VAR
	root : TOF_Core.CONFIGURATION_NODE;
	paramsNode : TOF_Core.CONFIGURATION_NODE;
	flagsNode : TOF_Core.CONFIGURATION_NODE;
	header : STRING(80) := 'test-structure';
	gain : REAL := 2.5;
	offset : DINT := 10;
	flag0 : BOOL := TRUE;
	flag1 : BOOL := FALSE;
	flag2 : BOOL := TRUE;
	headerDst : STRING(80);
	gainDst : REAL;
	offsetDst : DINT;
	flagDst : BOOL;
END_VAR
_Writer.BeginDocument();

// SA0175: Raw string buffer binding for header property; no character indexing.
{analysis -175}
_Writer.WriteValue(
	name := 'header',
	valueType := TOF_Core.CONFIGURATION_VALUE_TYPE.TYPE_STRING,
	data := ADR(header),
	size := SIZEOF(header)
);
{analysis +175}

_Writer.BeginObject(name := 'params');
_Writer.WriteValue(
	name := 'gain',
	valueType := TOF_Core.CONFIGURATION_VALUE_TYPE.TYPE_REAL,
	data := ADR(gain),
	size := SIZEOF(gain)
);
_Writer.WriteValue(
	name := 'offset',
	valueType := TOF_Core.CONFIGURATION_VALUE_TYPE.TYPE_DINT,
	data := ADR(offset),
	size := SIZEOF(offset)
);
_Writer.EndObject();

_Writer.BeginArray(name := 'flags');
_Writer.WriteValue(
	name := '',
	valueType := TOF_Core.CONFIGURATION_VALUE_TYPE.TYPE_BOOL,
	data := ADR(flag0),
	size := SIZEOF(flag0)
);
_Writer.WriteValue(
	name := '',
	valueType := TOF_Core.CONFIGURATION_VALUE_TYPE.TYPE_BOOL,
	data := ADR(flag1),
	size := SIZEOF(flag1)
);
_Writer.WriteValue(
	name := '',
	valueType := TOF_Core.CONFIGURATION_VALUE_TYPE.TYPE_BOOL,
	data := ADR(flag2),
	size := SIZEOF(flag2)
);
_Writer.EndArray();

_Writer.EndDocument(document := _Doc);

root := _Reader.Parse(document := _Doc);

// SA0175: Raw string buffer binding for header property; no character indexing.
{analysis -175}
_Reader.ReadValue(
	node := _Reader.GetField(node := root, name := 'header'),
	valueType := TOF_Core.CONFIGURATION_VALUE_TYPE.TYPE_STRING,
	data := ADR(headerDst),
	size := SIZEOF(headerDst)
);
{analysis +175}
Assert.ThatString(actual := headerDst).ToBe(expected := 'test-structure');

paramsNode := _Reader.GetField(node := root, name := 'params');
_Reader.ReadValue(
	node := _Reader.GetField(node := paramsNode, name := 'gain'),
	valueType := TOF_Core.CONFIGURATION_VALUE_TYPE.TYPE_REAL,
	data := ADR(gainDst),
	size := SIZEOF(gainDst)
);
Assert.ThatReal(actual := gainDst).ToBe(expected := 2.5, tolerance := 0.001);

_Reader.ReadValue(
	node := _Reader.GetField(node := paramsNode, name := 'offset'),
	valueType := TOF_Core.CONFIGURATION_VALUE_TYPE.TYPE_DINT,
	data := ADR(offsetDst),
	size := SIZEOF(offsetDst)
);
Assert.ThatDInt(actual := offsetDst).ToBe(expected := 10);

flagsNode := _Reader.GetField(node := root, name := 'flags');
Assert.ThatUDInt(actual := _Reader.GetArraySize(node := flagsNode)).ToBe(expected := 3);

_Reader.ReadValue(
	node := _Reader.GetItem(node := flagsNode, index := 0),
	valueType := TOF_Core.CONFIGURATION_VALUE_TYPE.TYPE_BOOL,
	data := ADR(flagDst),
	size := SIZEOF(flagDst)
);
Assert.ThatBool(actual := flagDst).IsTrue();

_Reader.ReadValue(
	node := _Reader.GetItem(node := flagsNode, index := 1),
	valueType := TOF_Core.CONFIGURATION_VALUE_TYPE.TYPE_BOOL,
	data := ADR(flagDst),
	size := SIZEOF(flagDst)
);
Assert.ThatBool(actual := flagDst).IsFalse();

_Reader.ReadValue(
	node := _Reader.GetItem(node := flagsNode, index := 2),
	valueType := TOF_Core.CONFIGURATION_VALUE_TYPE.TYPE_BOOL,
	data := ADR(flagDst),
	size := SIZEOF(flagDst)
);
Assert.ThatBool(actual := flagDst).IsTrue();
END_METHOD

(*!
<summary>Verifies empty, Unicode and escaped wide strings, including an independently encoded JSON escape.</summary>
<description>Checks that data following the wide null terminator is excluded from the serialized JSON string.</description>
*)
METHOD PRIVATE testWideStringsRoundTrip
VAR
	root : TOF_Core.CONFIGURATION_NODE;
	domRoot : Tc3_JsonXml.SJsonValue;
	emptyValue : Tc3_JsonXml.SJsonValue;
	emptyWide : WSTRING(80) := "";
	regWide : WSTRING(80) := "Café";
	escapeWide : WSTRING(80) := "Wide $N newline and \ backslash";
	wstrDst : WSTRING(80) := "initial";
END_VAR
emptyWide[1] := 16#0058; // Leave an X after the terminator to detect serialization of unused storage.

_Writer.BeginDocument();
_Writer.WriteValue(
	name := 'emptyWide',
	valueType := TOF_Core.CONFIGURATION_VALUE_TYPE.TYPE_WSTRING,
	data := ADR(emptyWide),
	size := SIZEOF(emptyWide)
);
_Writer.WriteValue(
	name := 'regWide',
	valueType := TOF_Core.CONFIGURATION_VALUE_TYPE.TYPE_WSTRING,
	data := ADR(regWide),
	size := SIZEOF(regWide)
);
_Writer.WriteValue(
	name := 'escapeWide',
	valueType := TOF_Core.CONFIGURATION_VALUE_TYPE.TYPE_WSTRING,
	data := ADR(escapeWide),
	size := SIZEOF(escapeWide)
);
_Writer.EndDocument(document := _Doc);

domRoot := _Dom.ParseDocument(sJson := _Doc);
emptyValue := _Dom.FindMember(v := domRoot, member := 'emptyWide');

IF emptyValue = 0 OR_ELSE NOT _Dom.IsString(v := emptyValue) THEN
	RecordFailure(message := "Writer did not emit emptyWide as a JSON string");
	RETURN;
END_IF

Assert.ThatUDInt(
	actual := _Dom.GetStringLength(v := emptyValue),
	message := "Serialized emptyWide contains only the terminator"
).ToBe(expected := TOF_Core.Strings.CharSize);

root := _Reader.Parse(document := _Doc);

_Reader.ReadValue(
	node := _Reader.GetField(node := root, name := 'emptyWide'),
	valueType := TOF_Core.CONFIGURATION_VALUE_TYPE.TYPE_WSTRING,
	data := ADR(wstrDst),
	size := SIZEOF(wstrDst)
);
Assert.ThatWideString(actual := wstrDst).ToBe(expected := "");

_Reader.ReadValue(
	node := _Reader.GetField(node := root, name := 'regWide'),
	valueType := TOF_Core.CONFIGURATION_VALUE_TYPE.TYPE_WSTRING,
	data := ADR(wstrDst),
	size := SIZEOF(wstrDst)
);
Assert.ThatWideString(actual := wstrDst).ToBe(expected := "Café");

_Reader.ReadValue(
	node := _Reader.GetField(node := root, name := 'escapeWide'),
	valueType := TOF_Core.CONFIGURATION_VALUE_TYPE.TYPE_WSTRING,
	data := ADR(wstrDst),
	size := SIZEOF(wstrDst)
);
Assert.ThatWideString(actual := wstrDst).ToBe(expected := "Wide $N newline and \ backslash");

_Doc := '{"unicode":"Caf\u00e9"}';
root := _Reader.Parse(document := _Doc);
wstrDst := "initial";
_Reader.ReadValue(
	node := _Reader.GetField(node := root, name := 'unicode'),
	valueType := TOF_Core.CONFIGURATION_VALUE_TYPE.TYPE_WSTRING,
	data := ADR(wstrDst),
	size := SIZEOF(wstrDst)
);
Assert.ThatWideString(actual := wstrDst, message := "Decode a JSON Unicode escape").ToBe(
	expected := "Café"
);
END_METHOD

END_FUNCTION_BLOCK

// ---- Tests/Devices/IO/RangeAnalogValueConverterTest.TcPOU
(*
SPDX-FileCopyrightText: c 2026 Oleksandr Tiutyk <trofimich@gmail.com>
SPDX-License-Identifier: MIT
License: https://opensource.org/license/mit
*)

(*!
<summary>Groups the three raw representations tested by the range converter suite.</summary>
<description>
Owns persistent child storage and fixed parent associations. Use in one task without reentry and do not copy the group.
Children is borrowed and must not be modified by application code. Constructor callbacks are not used.
</description>
*)

{attribute 'no_assign'}
{attribute 'no_explicit_call' := 'do not call this function block directly'}
FUNCTION_BLOCK RangeAnalogValueConverterTest EXTENDS TOF_Testing.TestGroup<3>
VAR_STAT
	{attribute 'hide'}
	_ClassName : STRING := __POUNAME();
END_VAR
VAR
	_Test16Bit : RangeAnalogValueConverter16BitTest(name := "Test16Bit", parent := THIS^);
	_Test32Bit : RangeAnalogValueConverter32BitTest(name := "Test32Bit", parent := THIS^);
	_Test32Real : RangeAnalogValueConverter32RealTest(name := "Test32Real", parent := THIS^);

	_Children : ARRAY [0.._ChildCount - 1] OF TOF_Testing.ITestElement :=
	[
		_Test16Bit,
		_Test32Bit,
		_Test32Real
	];
END_VAR

//! <summary>Borrows the fixed array of this concrete group; do not modify it.</summary>
{attribute 'monitoring' := 'call'}
PROPERTY Children : REFERENCE TO ARRAY [0.._ChildCount - 1] OF TOF_Testing.ITestElement
GET
Children REF= _Children;
END_GET
END_PROPERTY

//! <summary>Borrows the concrete class name for the lifetime of this instance; callers must not modify it.</summary>
{attribute 'monitoring' := 'call'}
PROPERTY ClassName : REFERENCE TO STRING
GET
ClassName REF= _ClassName;
END_GET
END_PROPERTY

//! <summary>Borrows the compiler-initialized namespace; callers must not modify the returned reference.</summary>
{attribute 'monitoring' := 'call'}
PROPERTY NamespaceName : REFERENCE TO STRING
GET
NamespaceName REF= CurrentNamespace.Name;
END_GET
END_PROPERTY

//! <summary>Reports the complete concrete instance size, excluding separately allocated storage.</summary>
{attribute 'monitoring' := 'call'}
PROPERTY SelfSize : ULINT
GET
SelfSize := XSIZEOF(THIS^);
END_GET
END_PROPERTY

END_FUNCTION_BLOCK

// ---- Tests/Devices/IO/RangeAnalogValueConverter16BitTest.TcPOU
(*
SPDX-FileCopyrightText: © 2026 Oleksandr Tiutyk <trofimich@gmail.com>
SPDX-License-Identifier: MIT
License: https://opensource.org/license/mit
*)

(*!
<summary>Checks 16-bit integer conversion on ascending and descending engineering scales.</summary>
<description>Verifies interpolation, saturation and the zeroed upper bytes of the raw result.</description>
*)

{attribute 'no_assign'}
{attribute 'no_explicit_call' := 'do not call this function block directly'}
FUNCTION_BLOCK RangeAnalogValueConverter16BitTest EXTENDS TOF_Testing.SingleCycleTest
VAR_STAT
	{attribute 'hide'}
	_ClassName : STRING := __POUNAME();
END_VAR

(*!
<summary>Borrows the concrete class name for the lifetime of this instance.</summary>
*)
{attribute 'monitoring' := 'call'}
PROPERTY ClassName : REFERENCE TO STRING
GET
ClassName REF= _ClassName;
END_GET
END_PROPERTY

(*!
<summary>Checks five ascending points in each direction and clamping and interpolation on the descending scale.</summary>
*)
METHOD PROTECTED ExecuteTest
VAR CONSTANT
	analogPoints : ARRAY [0..4] OF LREAL := [0, 2.5, 5, 7.5, 10];
	expectedRaw : ARRAY [0..4] OF INT := [TOF_Core.SignedInt16.MIN_VALUE, -16384, -1, 16383, TOF_Core.SignedInt16.MAX_VALUE];
	rawInputs : ARRAY [0..4] OF INT := [TOF_Core.SignedInt16.MIN_VALUE, -16384, 0, 16383, TOF_Core.SignedInt16.MAX_VALUE];
END_VAR
VAR
	i : DINT;
	zeroToTen : TOF_Devices_IO.StaticRangeAnalogValueConverter(
		minAnalogValue := 0,
		maxAnalogValue := 10,
		minRawValue := TOF_Devices_IO.RawAnalogValues.FromInt16(value := TOF_Core.SignedInt16.MIN_VALUE),
		maxRawValue := TOF_Devices_IO.RawAnalogValues.FromInt16(value := TOF_Core.SignedInt16.MAX_VALUE)
	);
	descendingEngineering : TOF_Devices_IO.StaticRangeAnalogValueConverter(
		minAnalogValue := 30,
		maxAnalogValue := -10,
		minRawValue := TOF_Devices_IO.RawAnalogValues.FromInt16(value := -200),
		maxRawValue := TOF_Devices_IO.RawAnalogValues.FromInt16(value := 600)
	);

	rawValue : TOF_Devices_IO.RAW_ANALOG_VALUE;
	analogValue : LREAL;
END_VAR
FOR i := LOWER_BOUND(analogPoints, 1) TO UPPER_BOUND(analogPoints, 1) DO
	rawValue := zeroToTen.ConvertAnalogValueToRawValue(
		analogValue := analogPoints[i],
		rawValueType := TOF_Devices_IO.RAW_ANALOG_VALUE_TYPE.INT16
	);
	Assert.ThatInt(
		actual := rawValue.Int16,
		message := TOF_Core.WideStrings.Concat255("Analog to raw at ", TO_WSTRING(analogPoints[i]))
	).ToBe(expected := expectedRaw[i]);

	analogValue := zeroToTen.ConvertRawValueToAnalogValue(
		rawValue := TOF_Devices_IO.RawAnalogValues.FromInt16(value := rawInputs[i]),
		rawValueType := TOF_Devices_IO.RAW_ANALOG_VALUE_TYPE.INT16
	);
	Assert.ThatLongReal(
		actual := analogValue,
		message := TOF_Core.WideStrings.Concat255("Raw to analog at ", TO_WSTRING(rawInputs[i]))
	).ToBe(expected := analogPoints[i], tolerance := 0.01);
END_FOR

rawValue := zeroToTen.ConvertAnalogValueToRawValue(
	analogValue := 2.5,
	rawValueType := TOF_Devices_IO.RAW_ANALOG_VALUE_TYPE.INT16
);
Assert.ThatDInt(actual := rawValue.Int32, message := "Negative INT16 results must have zero upper bytes").ToBe(
	expected := DINT#16#0000C000
);

// Check the descending scale independently of the ascending fixture.
rawValue := descendingEngineering.ConvertAnalogValueToRawValue(
	analogValue := 40,
	rawValueType := TOF_Devices_IO.RAW_ANALOG_VALUE_TYPE.INT16
);
Assert.ThatInt(
	actual := rawValue.Int16,
	message := "Analog to raw clamps above its first endpoint"
).ToBe(expected := -200);

rawValue := descendingEngineering.ConvertAnalogValueToRawValue(
	analogValue := 20,
	rawValueType := TOF_Devices_IO.RAW_ANALOG_VALUE_TYPE.INT16
);
Assert.ThatInt(
	actual := rawValue.Int16,
	message := "Analog to raw interpolates an interior value"
).ToBe(expected := 0);

rawValue := descendingEngineering.ConvertAnalogValueToRawValue(
	analogValue := -20,
	rawValueType := TOF_Devices_IO.RAW_ANALOG_VALUE_TYPE.INT16
);
Assert.ThatInt(
	actual := rawValue.Int16,
	message := "Analog to raw clamps below its last endpoint"
).ToBe(expected := 600);

analogValue := descendingEngineering.ConvertRawValueToAnalogValue(
	rawValue := TOF_Devices_IO.RawAnalogValues.FromInt16(value := -300),
	rawValueType := TOF_Devices_IO.RAW_ANALOG_VALUE_TYPE.INT16
);
Assert.ThatLongReal(
	actual := analogValue,
	message := "Raw to analog clamps below the raw minimum"
).ToBe(expected := 30);

analogValue := descendingEngineering.ConvertRawValueToAnalogValue(
	rawValue := TOF_Devices_IO.RawAnalogValues.FromInt16(value := 200),
	rawValueType := TOF_Devices_IO.RAW_ANALOG_VALUE_TYPE.INT16
);
Assert.ThatLongReal(
	actual := analogValue,
	message := "Raw to analog interpolates a descending engineering value"
).ToBe(expected := 10);

analogValue := descendingEngineering.ConvertRawValueToAnalogValue(
	rawValue := TOF_Devices_IO.RawAnalogValues.FromInt16(value := 700),
	rawValueType := TOF_Devices_IO.RAW_ANALOG_VALUE_TYPE.INT16
);
Assert.ThatLongReal(
	actual := analogValue,
	message := "Raw to analog clamps above the raw maximum"
).ToBe(expected := -10);
END_METHOD

(*!
<summary>Borrows the compiler-initialized namespace for the lifetime of this instance.</summary>
*)
{attribute 'monitoring' := 'call'}
PROPERTY NamespaceName : REFERENCE TO STRING
GET
NamespaceName REF= CurrentNamespace.Name;
END_GET
END_PROPERTY

(*!
<summary>Reports the complete concrete instance size in bytes.</summary>
*)
{attribute 'monitoring' := 'call'}
PROPERTY SelfSize : ULINT
GET
SelfSize := XSIZEOF(THIS^);
END_GET
END_PROPERTY

END_FUNCTION_BLOCK

// ---- Tests/Devices/IO/RangeAnalogValueConverter32BitTest.TcPOU
(*
SPDX-FileCopyrightText: © 2026 Oleksandr Tiutyk <trofimich@gmail.com>
SPDX-License-Identifier: MIT
License: https://opensource.org/license/mit
*)

(*!
<summary>Checks integer conversion on a 24-bit scale and a descending raw scale that uses more than 24 bits.</summary>
<description>Verifies interpolation, raw saturation and preservation of the 32-bit representation.</description>
*)

{attribute 'no_assign'}
{attribute 'no_explicit_call' := 'do not call this function block directly'}
FUNCTION_BLOCK RangeAnalogValueConverter32BitTest EXTENDS TOF_Testing.SingleCycleTest
VAR_STAT
	{attribute 'hide'}
	_ClassName : STRING := __POUNAME();
END_VAR

(*!
<summary>Borrows the concrete class name for the lifetime of this instance.</summary>
*)
{attribute 'monitoring' := 'call'}
PROPERTY ClassName : REFERENCE TO STRING
GET
ClassName REF= _ClassName;
END_GET
END_PROPERTY

(*!
<summary>Checks five ascending points in each direction and clamping and interpolation on the descending scale.</summary>
*)
METHOD PROTECTED ExecuteTest
VAR CONSTANT
	analogPoints : ARRAY [0..4] OF LREAL := [0, 2.5, 5, 7.5, 10];
	expectedRaw : ARRAY [0..4] OF DINT := [
		TOF_Core.SignedInt32.MIN_24BIT_VALUE, -4194304, -1, 4194303, TOF_Core.SignedInt32.MAX_24BIT_VALUE
	];
	rawInputs : ARRAY [0..4] OF DINT := [
		TOF_Core.SignedInt32.MIN_24BIT_VALUE, -4194304, 0, 4194304, TOF_Core.SignedInt32.MAX_24BIT_VALUE
	];
END_VAR
VAR
	i : DINT;
	zeroToTen : TOF_Devices_IO.StaticRangeAnalogValueConverter(
		minAnalogValue := 0,
		maxAnalogValue := 10,
		minRawValue := TOF_Devices_IO.RawAnalogValues.FromInt32(value := TOF_Core.SignedInt32.MIN_24BIT_VALUE),
		maxRawValue := TOF_Devices_IO.RawAnalogValues.FromInt32(value := TOF_Core.SignedInt32.MAX_24BIT_VALUE)
	);
	descendingRaw : TOF_Devices_IO.StaticRangeAnalogValueConverter(
		minAnalogValue := -10,
		maxAnalogValue := 30,
		minRawValue := TOF_Devices_IO.RawAnalogValues.FromInt32(value := 20000000),
		maxRawValue := TOF_Devices_IO.RawAnalogValues.FromInt32(value := -12000000)
	);

	rawValue : TOF_Devices_IO.RAW_ANALOG_VALUE;
	analogValue : LREAL;
END_VAR
FOR i := LOWER_BOUND(analogPoints, 1) TO UPPER_BOUND(analogPoints, 1) DO
	rawValue := zeroToTen.ConvertAnalogValueToRawValue(
		analogValue := analogPoints[i],
		rawValueType := TOF_Devices_IO.RAW_ANALOG_VALUE_TYPE.INT32
	);
	Assert.ThatDInt(
		actual := rawValue.Int32,
		message := TOF_Core.WideStrings.Concat255("Analog to raw at ", TO_WSTRING(analogPoints[i]))
	).ToBe(expected := expectedRaw[i]);

	analogValue := zeroToTen.ConvertRawValueToAnalogValue(
		rawValue := TOF_Devices_IO.RawAnalogValues.FromInt32(value := rawInputs[i]),
		rawValueType := TOF_Devices_IO.RAW_ANALOG_VALUE_TYPE.INT32
	);
	Assert.ThatLongReal(
		actual := analogValue,
		message := TOF_Core.WideStrings.Concat255("Raw to analog at ", TO_WSTRING(rawInputs[i]))
	).ToBe(expected := analogPoints[i], tolerance := 0.01);
END_FOR

// Check the descending scale independently of the ascending fixture.
rawValue := descendingRaw.ConvertAnalogValueToRawValue(
	analogValue := -20,
	rawValueType := TOF_Devices_IO.RAW_ANALOG_VALUE_TYPE.INT32
);
Assert.ThatDInt(
	actual := rawValue.Int32,
	message := "Analog to raw clamps to its first raw endpoint"
).ToBe(expected := 20000000);

rawValue := descendingRaw.ConvertAnalogValueToRawValue(
	analogValue := 0,
	rawValueType := TOF_Devices_IO.RAW_ANALOG_VALUE_TYPE.INT32
);
Assert.ThatDInt(
	actual := rawValue.Int32,
	message := "Analog to raw preserves values beyond 24 bits"
).ToBe(expected := 12000000);

rawValue := descendingRaw.ConvertAnalogValueToRawValue(
	analogValue := 40,
	rawValueType := TOF_Devices_IO.RAW_ANALOG_VALUE_TYPE.INT32
);
Assert.ThatDInt(
	actual := rawValue.Int32,
	message := "Analog to raw clamps to its last raw endpoint"
).ToBe(expected := -12000000);

analogValue := descendingRaw.ConvertRawValueToAnalogValue(
	rawValue := TOF_Devices_IO.RawAnalogValues.FromInt32(value := 21000000),
	rawValueType := TOF_Devices_IO.RAW_ANALOG_VALUE_TYPE.INT32
);
Assert.ThatLongReal(
	actual := analogValue,
	message := "Raw to analog clamps above the first raw endpoint"
).ToBe(expected := -10);

analogValue := descendingRaw.ConvertRawValueToAnalogValue(
	rawValue := TOF_Devices_IO.RawAnalogValues.FromInt32(value := -4000000),
	rawValueType := TOF_Devices_IO.RAW_ANALOG_VALUE_TYPE.INT32
);
Assert.ThatLongReal(
	actual := analogValue,
	message := "Raw to analog interpolates a descending raw value"
).ToBe(expected := 20);

analogValue := descendingRaw.ConvertRawValueToAnalogValue(
	rawValue := TOF_Devices_IO.RawAnalogValues.FromInt32(value := -13000000),
	rawValueType := TOF_Devices_IO.RAW_ANALOG_VALUE_TYPE.INT32
);
Assert.ThatLongReal(
	actual := analogValue,
	message := "Raw to analog clamps below the last raw endpoint"
).ToBe(expected := 30);
END_METHOD

(*!
<summary>Borrows the compiler-initialized namespace for the lifetime of this instance.</summary>
*)
{attribute 'monitoring' := 'call'}
PROPERTY NamespaceName : REFERENCE TO STRING
GET
NamespaceName REF= CurrentNamespace.Name;
END_GET
END_PROPERTY

(*!
<summary>Reports the complete concrete instance size in bytes.</summary>
*)
{attribute 'monitoring' := 'call'}
PROPERTY SelfSize : ULINT
GET
SelfSize := XSIZEOF(THIS^);
END_GET
END_PROPERTY

END_FUNCTION_BLOCK

// ---- Tests/Devices/IO/RangeAnalogValueConverter32RealTest.TcPOU
(*
SPDX-FileCopyrightText: © 2026 Oleksandr Tiutyk <trofimich@gmail.com>
SPDX-License-Identifier: MIT
License: https://opensource.org/license/mit
*)

(*!
<summary>Checks asymmetric fractional REAL32 scaling in both directions.</summary>
<description>All expected values are exact binary fractions. The inputs expose unintended integer conversion.</description>
*)

{attribute 'no_assign'}
{attribute 'no_explicit_call' := 'do not call this function block directly'}
FUNCTION_BLOCK RangeAnalogValueConverter32RealTest EXTENDS TOF_Testing.SingleCycleTest
VAR_STAT
	{attribute 'hide'}
	_ClassName : STRING := __POUNAME();
END_VAR

(*!
<summary>Borrows the concrete class name for the lifetime of this instance.</summary>
*)
{attribute 'monitoring' := 'call'}
PROPERTY ClassName : REFERENCE TO STRING
GET
ClassName REF= _ClassName;
END_GET
END_PROPERTY

(*!
<summary>Checks fixed interpolation and clamping expectations in both conversion directions.</summary>
*)
METHOD PROTECTED ExecuteTest
VAR
	fractionalRaw : TOF_Devices_IO.StaticRangeAnalogValueConverter(
		minAnalogValue := -4,
		maxAnalogValue := 12,
		minRawValue := TOF_Devices_IO.RawAnalogValues.FromReal32(value := -2.75),
		maxRawValue := TOF_Devices_IO.RawAnalogValues.FromReal32(value := 1.75)
	);

	rawValue : TOF_Devices_IO.RAW_ANALOG_VALUE;
	analogValue : LREAL;
END_VAR
rawValue := fractionalRaw.ConvertAnalogValueToRawValue(
	analogValue := -8,
	rawValueType := TOF_Devices_IO.RAW_ANALOG_VALUE_TYPE.REAL32
);
Assert.ThatReal(
	actual := rawValue.Real32,
	message := "Analog to raw clamps below its engineering minimum"
).ToBe(expected := -2.75);

rawValue := fractionalRaw.ConvertAnalogValueToRawValue(
	analogValue := 2,
	rawValueType := TOF_Devices_IO.RAW_ANALOG_VALUE_TYPE.REAL32
);
Assert.ThatReal(
	actual := rawValue.Real32,
	message := "Analog to raw preserves fractional interpolation"
).ToBe(expected := -1.0625);

rawValue := fractionalRaw.ConvertAnalogValueToRawValue(
	analogValue := 8,
	rawValueType := TOF_Devices_IO.RAW_ANALOG_VALUE_TYPE.REAL32
);
Assert.ThatReal(
	actual := rawValue.Real32,
	message := "Analog to raw preserves positive fractional interpolation"
).ToBe(expected := 0.625);

rawValue := fractionalRaw.ConvertAnalogValueToRawValue(
	analogValue := 16,
	rawValueType := TOF_Devices_IO.RAW_ANALOG_VALUE_TYPE.REAL32
);
Assert.ThatReal(
	actual := rawValue.Real32,
	message := "Analog to raw clamps above its engineering maximum"
).ToBe(expected := 1.75);

analogValue := fractionalRaw.ConvertRawValueToAnalogValue(
	rawValue := TOF_Devices_IO.RawAnalogValues.FromReal32(value := -3),
	rawValueType := TOF_Devices_IO.RAW_ANALOG_VALUE_TYPE.REAL32
);
Assert.ThatLongReal(
	actual := analogValue,
	message := "Raw to analog clamps below the fractional raw minimum"
).ToBe(expected := -4);

analogValue := fractionalRaw.ConvertRawValueToAnalogValue(
	rawValue := TOF_Devices_IO.RawAnalogValues.FromReal32(value := -1.0625),
	rawValueType := TOF_Devices_IO.RAW_ANALOG_VALUE_TYPE.REAL32
);
Assert.ThatLongReal(
	actual := analogValue,
	message := "Raw to analog preserves the fractional raw input"
).ToBe(expected := 2);

analogValue := fractionalRaw.ConvertRawValueToAnalogValue(
	rawValue := TOF_Devices_IO.RawAnalogValues.FromReal32(value := 0.625),
	rawValueType := TOF_Devices_IO.RAW_ANALOG_VALUE_TYPE.REAL32
);
Assert.ThatLongReal(
	actual := analogValue,
	message := "Raw to analog preserves the positive fractional raw input"
).ToBe(expected := 8);

analogValue := fractionalRaw.ConvertRawValueToAnalogValue(
	rawValue := TOF_Devices_IO.RawAnalogValues.FromReal32(value := 2),
	rawValueType := TOF_Devices_IO.RAW_ANALOG_VALUE_TYPE.REAL32
);
Assert.ThatLongReal(
	actual := analogValue,
	message := "Raw to analog clamps above the fractional raw maximum"
).ToBe(expected := 12);
END_METHOD

(*!
<summary>Borrows the compiler-initialized namespace for the lifetime of this instance.</summary>
*)
{attribute 'monitoring' := 'call'}
PROPERTY NamespaceName : REFERENCE TO STRING
GET
NamespaceName REF= CurrentNamespace.Name;
END_GET
END_PROPERTY

(*!
<summary>Reports the complete concrete instance size in bytes.</summary>
*)
{attribute 'monitoring' := 'call'}
PROPERTY SelfSize : ULINT
GET
SelfSize := XSIZEOF(THIS^);
END_GET
END_PROPERTY

END_FUNCTION_BLOCK

// ---- Tests/Tasks/Stopping/TimerRestartWhileRunningTest.TcPOU
(*
SPDX-FileCopyrightText: © 2026 Oleksandr Tiutyk <trofimich@gmail.com>
SPDX-License-Identifier: MIT
License: https://opensource.org/license/mit
*)

(*!
<summary>Checks a zero-interval restart of a running timer across two consecutive task cycles.</summary>
<description>
The first body call starts and restarts the timer. The next call observes completion.
Use in one cyclic task. Teardown prepares the owned timer for another run.
</description>
*)

{attribute 'no_explicit_call' := 'do not call this function block directly'}
FUNCTION_BLOCK TimerRestartWhileRunningTest EXTENDS TOF_Testing.MultiCycleTest
VAR
	_Timer : TOF_Timers.Timer(name := "timer");
END_VAR
VAR CONSTANT
	//! <summary>Keeps the first run active until the explicit restart.</summary>
	_ActiveInterval : TIME := T#1H;
END_VAR
VAR_STAT
	//! <summary>Class name shared by all instances of this function block.</summary>
	{attribute 'hide'}
	_ClassName : STRING := __POUNAME();
END_VAR
VAR
	{attribute 'hide'}
	{attribute 'init_namespace'}
	_NamespaceName : STRING;
END_VAR

(*!
<summary>Resets the timer after completion or failure.</summary>
*)
METHOD PROTECTED AfterTest
IF _Timer.State.Running THEN
	Assert.ThatBool(actual := _Timer.Cancel(), message := "Timer cleanup must accept cancellation").IsTrue();
	_Timer.Execute();
END_IF

IF _Timer.State.Stopped THEN
	Assert.ThatBool(actual := _Timer.Reset(), message := "Timer cleanup must accept Reset").IsTrue();
END_IF

Assert.ThatBool(actual := _Timer.State.Ready, message := "Timer must be ready for another run").IsTrue();
END_METHOD

//! <summary>Borrows the concrete class name for the lifetime of this instance; callers must not modify it.</summary>
{attribute 'monitoring' := 'call'}
PROPERTY ClassName : REFERENCE TO STRING
GET
ClassName REF= _ClassName;
END_GET
END_PROPERTY

(*!
<summary>Restarts the active timer in the first cycle and checks the completion pulse in the next.</summary>
<description>A refused start ends the scenario immediately. The framework invokes AfterTest even after failure.</description>
*)
METHOD PROTECTED ExecuteTest : TOF_Testing.TEST_CYCLE_RESULT
VAR
	restartAccepted : BOOL;
END_VAR
IF CycleCount = 1 THEN
	_Timer.Interval := _ActiveInterval;

	IF NOT _Timer.Start() THEN
		RecordFailure(message := "Prepared timer must accept Start");

		ExecuteTest := TOF_Testing.TEST_CYCLE_RESULT.DONE;
		RETURN;
	END_IF

	_Timer.Execute();
	Assert.ThatBool(
		actual := _Timer.State.Running,
		message := "Long interval must still be running before restart"
	).IsTrue();

	restartAccepted := _Timer.SetIntervalAndRestart(interval := TOF_Core.Times.MIN_VALUE);
	Assert.ThatBool(
		actual := restartAccepted,
		message := "Active restart must complete in the same cycle"
	).IsTrue();

	IF NOT restartAccepted THEN
		ExecuteTest := TOF_Testing.TEST_CYCLE_RESULT.DONE;
		RETURN;
	END_IF

	Assert.ThatBool(
		actual := _Timer.State.Running,
		message := "New zero interval must already be started"
	).IsTrue();
	Assert.ThatBool(
		actual := _Timer.Elapsed,
		message := "Zero interval first evaluates TON in Execute"
	).IsFalse();
	Assert.ThatBool(
		actual := _Timer.Triggered,
		message := "Restart itself must not retain a pulse"
	).IsFalse();

	ExecuteTest := TOF_Testing.TEST_CYCLE_RESULT.BUSY;
	RETURN;
END_IF

_Timer.Execute();
Assert.ThatBool(
	actual := _Timer.Elapsed,
	message := "Zero interval must immediately set TON.Q"
).IsTrue();
Assert.ThatBool(
	actual := _Timer.Triggered,
	message := "Restarted zero interval must trigger without another cycle"
).IsTrue();
Assert.ThatBool(
	actual := _Timer.State.Stopped,
	message := "Restarted timer must complete in that same Execute"
).IsTrue();
Assert.ThatBool(
	actual := _Timer.FinalStopReason.WorkDone,
	message := "Restarted timer must complete normally"
).IsTrue();

ExecuteTest := TOF_Testing.TEST_CYCLE_RESULT.DONE;
END_METHOD

//! <summary>Borrows the compiler-initialized namespace; callers must not modify the returned reference.</summary>
{attribute 'monitoring' := 'call'}
PROPERTY NamespaceName : REFERENCE TO STRING
GET
NamespaceName REF= CurrentNamespace.Name;
END_GET
END_PROPERTY

//! <summary>Reports the complete concrete instance size, excluding separately allocated storage.</summary>
{attribute 'monitoring' := 'call'}
PROPERTY SelfSize : ULINT
GET
SelfSize := XSIZEOF(THIS^);
END_GET
END_PROPERTY

END_FUNCTION_BLOCK

// ---- Tests/Files/OpenMissingFileForReadingTest.TcPOU
(*
SPDX-FileCopyrightText: © 2026 Oleksandr Tiutyk <trofimich@gmail.com>
SPDX-License-Identifier: MIT
License: https://opensource.org/license/mit
*)

(*!
<summary>Checks resource acquisition failure when reading a missing file in an owned test directory.</summary>
<description>
The shared FileTestRoot is driven by the test controller. This instance owns its directory and file tasks
for the entire scenario. The ten-second scenario deadline excludes cleanup. Setup or scenario failures
are retained while the manager stops and the directory cleanup attempts finish. Only then is a result
reported. Native failures can leave artifacts requiring inspection. Use from one task without reentry.
Do not copy the instance or drive borrowed file tasks independently.
</description>
*)

{attribute 'no_assign'}
{attribute 'no_explicit_call' := 'do not call this function block directly'}
FUNCTION_BLOCK OpenMissingFileForReadingTest EXTENDS TOF_Testing.TestCase
VAR CONSTANT
	//! <summary>Bounds scenario preparation and execution before cleanup is requested.</summary>
	_ScenarioTimeout : TIME := T#10S;
	//! <summary>FB_FileOpen code for a missing file or invalid filename or path.</summary>
	_FileNotFoundCode : UDINT := 16#70C;
END_VAR
VAR
	_Directory : FileTestDirectory(directoryPath := 'C:\OpenFrameworkTests\FileContent_Missing');
	_FileContentManager : TOF_FileSystem.FileContentManager(name := "fileContentManager");
	_ReadStringFromFile : TOF_FileSystem.ReadString255FromFile(name := "readStringFromFile");
	_ScenarioDeadline : Tc2_Standard.TON;

	_Lifecycle : FILE_TEST_LIFECYCLE;
	_ScenarioFailure : TOF_Core.ERROR_MESSAGE;
	_CleanupExceptionObserved : BOOL;
END_VAR
VAR_STAT
	//! <summary>Class name shared by all instances of this function block.</summary>
	{attribute 'hide'}
	_ClassName : STRING := __POUNAME();
END_VAR
VAR
	{attribute 'hide'}
	{attribute 'init_namespace'}
	_NamespaceName : STRING;
END_VAR

(*!
<summary>Prepares the owned fixture and file queue for a fresh run.</summary>
<description>
After a previous run, reuse requires successful directory cleanup and idle file tasks. If a reset is refused,
report failure without submitting new native I/O. A retained resource requires inspection before reuse.
</description>
*)
METHOD PROTECTED BeforeTest
IF _Lifecycle = FILE_TEST_LIFECYCLE.FINISHED THEN
	IF _FileContentManager.State.Running
		OR_ELSE _FileContentManager.ResourceManager.ResourceAcquired
		OR_ELSE NOT _FileContentManager.Reset()
	THEN
		RecordFailure(message := "Missing-file fixture could not be rearmed after the previous run");
		RETURN;
	END_IF

	// Reset on a READY manager does not clear its queue after a refused Start.
	_FileContentManager.ClearWaitingTasks();

	IF NOT _ReadStringFromFile.Reset() OR_ELSE NOT _Directory.Reset() THEN
		RecordFailure(message := "Missing-file directory or read task could not be rearmed after the previous run");
		RETURN;
	END_IF
END_IF

_ScenarioDeadline(IN := FALSE, PT := _ScenarioTimeout);
_ScenarioFailure := "";
_CleanupExceptionObserved := FALSE;
_Lifecycle := FILE_TEST_LIFECYCLE.RUNNING_SCENARIO;
END_METHOD

//! <summary>Borrows the concrete class name for the lifetime of this instance; callers must not modify it.</summary>
{attribute 'monitoring' := 'call'}
PROPERTY ClassName : REFERENCE TO STRING
GET
ClassName REF= _ClassName;
END_GET
END_PROPERTY

(*!
<summary>Advances the scenario or one cycle of cleanup before publishing its result.</summary>
<description>
Retains an ordinary scenario failure without calling RecordFailure until cleanup completes, because that
call ends the leaf after this callback. A caught cleanup exception keeps the persistent fixture available
for another attempt on the next cycle. The inherited test boundary handles terminal allocation failure.
</description>
*)
METHOD PROTECTED RunCycle : TOF_Testing.TEST_CYCLE_RESULT
VAR
	cleanupFailure : WSTRING(255);
END_VAR
RunCycle := TOF_Testing.TEST_CYCLE_RESULT.BUSY;

IF _Lifecycle = FILE_TEST_LIFECYCLE.RUNNING_SCENARIO THEN
	__TRY
		IF runScenario() THEN
			_Lifecycle := FILE_TEST_LIFECYCLE.CLEANING_UP;
		END_IF
	__CATCH
		_ScenarioFailure := "Exception interrupted the file scenario";
		_Lifecycle := FILE_TEST_LIFECYCLE.CLEANING_UP;
	__ENDTRY

	RETURN;
END_IF

__TRY
	IF _FileContentManager.State.Running THEN
		_FileContentManager.Cancel();
		_FileContentManager.Execute();

		IF _FileContentManager.State.Running THEN
			RETURN;
		END_IF
	END_IF

	_Directory.Cleanup();
__CATCH
	_CleanupExceptionObserved := TRUE;
	RETURN;
__ENDTRY

IF NOT _Directory.CleanupComplete THEN
	RETURN;
END_IF

IF NOT _Directory.CleanupSucceeded THEN
	cleanupFailure := TOF_Core.WideStrings.ConcatFit255(
		"Cleanup failed for ", TO_WSTRING(_Directory.DirectoryPath), ": ", TO_WSTRING(_Directory.CleanupMessage)
	);
ELSIF _CleanupExceptionObserved THEN
	cleanupFailure := "An exception interrupted cleanup before the final removal attempt";
END_IF

IF cleanupFailure <> "" THEN
	IF _ScenarioFailure <> "" THEN
		TOF_Core.WideStrings.AppendFit(targetString := _ScenarioFailure, sourceString := " | ");
	END_IF

	TOF_Core.WideStrings.AppendFit(targetString := _ScenarioFailure, sourceString := cleanupFailure);
END_IF

IF _ScenarioFailure <> "" THEN
	RecordFailure(message := _ScenarioFailure);
END_IF

_Lifecycle := FILE_TEST_LIFECYCLE.FINISHED;
RunCycle := TOF_Testing.TEST_CYCLE_RESULT.DONE;
END_METHOD

(*!
<summary>Advances directory preparation and verifies the expected failure to acquire a read handle.</summary>
<description>
Returns TRUE once the scenario has passed or a failure requires cleanup. Copies the first failed
expectation, leaving reporting to RunCycle after cleanup. The expected open diagnostic identifies the exact
file in the newly created directory and its native code. Waiting for the shared root counts toward the same scenario deadline.
</description>
*)
METHOD PRIVATE runScenario : BOOL
VAR
	expectedOpenFailure : TOF_Core.ERROR_MESSAGE;
END_VAR
_ScenarioDeadline(IN := TRUE, PT := _ScenarioTimeout);

IF FileTestRoot.FailureMessage <> TOF_Core.Strings.Empty THEN
	_ScenarioFailure := TO_WSTRING(FileTestRoot.FailureMessage);
	runScenario := TRUE;
	RETURN;
END_IF

IF NOT FileTestRoot.Prepared THEN
	IF _ScenarioDeadline.Q THEN
		_ScenarioFailure := "Shared filesystem test root was not ready within 10 seconds";
		runScenario := TRUE;
	END_IF

	RETURN;
END_IF

_Directory.Prepare();

IF _Directory.PreparationFailed THEN
	_ScenarioFailure := TOF_Core.WideStrings.ConcatFit255(
		TO_WSTRING(_Directory.DirectoryPath), ": ", TO_WSTRING(_Directory.PreparationMessage)
	);
	runScenario := TRUE;
	RETURN;
END_IF

IF NOT _Directory.Prepared THEN
	IF _ScenarioDeadline.Q THEN
		_ScenarioFailure := "Scenario directory preparation exceeded its deadline";
		runScenario := TRUE;
	END_IF

	RETURN;
END_IF

IF _FileContentManager.State.Ready THEN
	_FileContentManager.FilePath := _Directory.FirstFilePath;
	_FileContentManager.ModeFlags := Tc2_System.Global_Variables.FOPEN_MODEREAD
		OR Tc2_System.Global_Variables.FOPEN_MODETEXT;
	_FileContentManager.PathType := Tc2_System.E_OpenPath.PATH_GENERIC;
	_FileContentManager.Timeout := T#2S;
	_FileContentManager.StopWhenNoPendingTasks := TRUE;
	_FileContentManager.Enqueue(fileHandleTask := _ReadStringFromFile);

	IF NOT _FileContentManager.Start() THEN
		_ScenarioFailure := "Start must accept the task; the missing file must be detected during resource acquisition";
		runScenario := TRUE;
		RETURN;
	END_IF
END_IF

_FileContentManager.Execute();

IF _FileContentManager.State.Stopped THEN
	expectedOpenFailure := TOF_Core.WideStrings.Concat255(
		"Error while open file '",
		TO_WSTRING(_Directory.FirstFilePath),
		"'",
		TOF_Core.Exceptions.ERROR_CODE_PREFIX,
		TO_WSTRING(_FileNotFoundCode)
	);

	IF NOT _FileContentManager.FinalStopReason.Failure THEN
		_ScenarioFailure := "Opening a missing file for reading must stop FileContentManager with Failure";
	ELSIF _FileContentManager.FinalStopReason.Message <> expectedOpenFailure THEN
		_ScenarioFailure := "Expected the missing-file open error. Actual: ";
		TOF_Core.WideStrings.AppendFit(
			targetString := _ScenarioFailure,
			sourceString := _FileContentManager.FinalStopReason.Message
		);
	ELSIF NOT _ReadStringFromFile.State.Ready THEN
		_ScenarioFailure := "Read task must remain READY when the file cannot be opened";
	ELSIF _FileContentManager.ResourceManager.ResourceAcquired THEN
		_ScenarioFailure := "No file resource must remain acquired after file open failure";
	END_IF

	runScenario := TRUE;
ELSIF _ScenarioDeadline.Q THEN
	_ScenarioFailure := "FileContentManager did not stop within 10 seconds after attempting to open a missing file";
	runScenario := TRUE;
END_IF
END_METHOD

//! <summary>Borrows the compiler-initialized namespace; callers must not modify the returned reference.</summary>
{attribute 'monitoring' := 'call'}
PROPERTY NamespaceName : REFERENCE TO STRING
GET
NamespaceName REF= CurrentNamespace.Name;
END_GET
END_PROPERTY

//! <summary>Reports the complete concrete instance size, excluding separately allocated storage.</summary>
{attribute 'monitoring' := 'call'}
PROPERTY SelfSize : ULINT
GET
SelfSize := XSIZEOF(THIS^);
END_GET
END_PROPERTY

END_FUNCTION_BLOCK

// ---- Tests/Files/FileTestDirectory.TcPOU
(*
SPDX-FileCopyrightText: © 2026 Oleksandr Tiutyk <trofimich@gmail.com>
SPDX-License-Identifier: MIT
License: https://opensource.org/license/mit
*)

(*!
<summary>Owns preparation and nonrecursive cleanup of one filesystem test scenario directory.</summary>
<description>
The caller supplies a fixed path below the reserved test root and waits for FileTestRoot.Prepared before
Prepare. Ordinary creation must succeed before files may be registered or opened. Existing entries are not
adopted or deleted. One owner task drives the fixture and prevents external changes inside its directory.
Keep this instance alive and drain all scenario managers before Cleanup. Only registered fixed artifacts are
deleted. Failed or cancelled creation has unknown effects and grants no ownership; inspect that path manually.
Cleanup continues over later calls without a forced deadline. CleanupComplete reports completed attempts;
CleanupSucceeded reports directory removal or that creation was never submitted, not physical handle closure.
Reset can rearm a successfully cleaned fixture for another run.
</description>
*)

{attribute 'no_explicit_call' := 'Use Prepare and Cleanup from the owning scenario'}
FUNCTION_BLOCK FileTestDirectory
VAR
	_DirectoryPath : STRING(255);
	_Phase : FILE_TEST_DIRECTORY_PHASE;
	_OwnsDirectory : BOOL;
	_PreparationFailed : BOOL;
	_PreparationMessage : STRING(255);
	_CleanupComplete : BOOL;
	_CleanupSucceeded : BOOL;
	_CleanupMessage : STRING(255);
	_FirstFileMayExist : BOOL;
	_SecondFileMayExist : BOOL;

	_CreateDirectory : TOF_FileSystem.CreateDirectory(name := "prepareFileScenarioDirectory");
	_DeleteFirstFile : TOF_FileSystem.DeleteFile(name := "deleteFirstScenarioFile");
	_DeleteSecondFile : TOF_FileSystem.DeleteFile(name := "deleteSecondScenarioFile");
	_RemoveDirectory : TOF_FileSystem.RemoveEmptyDirectory(name := "removeFileScenarioDirectory");
END_VAR

(*!
<summary>Copies the fixed scenario directory path without performing I/O.</summary>
<description>
The caller supplies a path below C:\OpenFrameworkTests with enough room for the fixed artifact names.
The path remains unchanged throughout preparation, scenario execution and cleanup.
</description>
<param name="directoryPath">Fixed exclusively reserved scenario path below the prepared test root.</param>
*)
METHOD FB_init : BOOL
VAR_INPUT
	bInitRetains : BOOL; // TRUE: the retain variables are initialized (reset warm / reset cold)
	bInCopyCode : BOOL; // TRUE: the instance will be copied to the copy code afterward (online change)
	directoryPath : STRING(255);
END_VAR
IF NOT bInCopyCode THEN
	_DirectoryPath := directoryPath;
END_IF
END_METHOD

(*!
<summary>Advances ordinary directory creation and records ownership only after WORK_DONE.</summary>
<description>
Call only after the shared root is prepared. A refusal, native failure or caught exception reports preparation
failure. Keep invoking Cleanup after a failed scenario to drain an interrupted create; no existing entry is
adopted. Prepared remains FALSE until creation completes successfully.
</description>
*)
METHOD Prepare
__TRY

	CASE _Phase OF
		FILE_TEST_DIRECTORY_PHASE.CREATE_DIRECTORY:
			_CreateDirectory.DirectoryPath := _DirectoryPath;
			_CreateDirectory.PathType := Tc2_System.E_OpenPath.PATH_GENERIC;
			_CreateDirectory.Timeout := T#2S;

			IF _CreateDirectory.Start() THEN
				_Phase := FILE_TEST_DIRECTORY_PHASE.WAIT_FOR_DIRECTORY;
			ELSE
				_PreparationFailed := TRUE;
				_PreparationMessage := 'Scenario directory creation: Start refused';
				_Phase := FILE_TEST_DIRECTORY_PHASE.COMPLETE;
				_CleanupComplete := TRUE;
				_CleanupSucceeded := TRUE;
			END_IF

		FILE_TEST_DIRECTORY_PHASE.WAIT_FOR_DIRECTORY:
			_CreateDirectory.Execute();

			IF _CreateDirectory.State.Stopped THEN

				IF _CreateDirectory.FinalStopReason.WorkDone THEN
					_OwnsDirectory := TRUE;
					_Phase := FILE_TEST_DIRECTORY_PHASE.READY;
				ELSE
					_PreparationFailed := TRUE;
					_PreparationMessage := TO_STRING(_CreateDirectory.FinalStopReason.Message);
					_CleanupMessage := 'Creation failed; the scenario path is not owned and requires inspection';
					_Phase := FILE_TEST_DIRECTORY_PHASE.COMPLETE;
					_CleanupComplete := TRUE;
				END_IF

			END_IF

	END_CASE

__CATCH
	_PreparationFailed := TRUE;
	_PreparationMessage := 'Exception interrupted scenario directory creation';
__ENDTRY
END_METHOD

(*!
<summary>Registers the first fixed artifact before a scenario may create it.</summary>
<description>
Requires a successfully prepared, exclusively owned directory. Registration grants permission to attempt
cleanup of this fixed path even if a later open fails; it does not prove that the file exists.
</description>
*)
METHOD ExpectFirstFile
IF NOT _OwnsDirectory OR_ELSE _Phase <> FILE_TEST_DIRECTORY_PHASE.READY THEN
	TOF_Core.Exceptions.ThrowStandard(
		sourceNamespaceName := 'Tests',
		sourceClassName := 'FileTestDirectory',
		sourcePOUName := __POUNAME(),
		sourcePosition := __POSITION(),
		message := "A file artifact requires an owned prepared scenario directory"
	);
END_IF

_FirstFileMayExist := TRUE;
END_METHOD

(*!
<summary>Registers the second fixed artifact before a scenario may create it.</summary>
<description>
Requires a successfully prepared, exclusively owned directory. Registration grants permission to attempt
cleanup of this fixed path even if a later open fails; it does not prove that the file exists.
</description>
*)
METHOD ExpectSecondFile
IF NOT _OwnsDirectory OR_ELSE _Phase <> FILE_TEST_DIRECTORY_PHASE.READY THEN
	TOF_Core.Exceptions.ThrowStandard(
		sourceNamespaceName := 'Tests',
		sourceClassName := 'FileTestDirectory',
		sourcePOUName := __POUNAME(),
		sourcePosition := __POSITION(),
		message := "A file artifact requires an owned prepared scenario directory"
	);
END_IF

_SecondFileMayExist := TRUE;
END_METHOD

(*!
<summary>Drains preparation and attempts deletion of registered artifacts and the owned directory.</summary>
<description>
All scenario file managers and content tasks must already have completed stopping/release. Repeated calls
advance one cleanup phase without starting scenario I/O. A missing registered file can cause a deletion error;
successful final directory removal still proves that no artifact remains there. CleanupMessage retains any
intermediate error. No recursive deletion, adoption of existing directories or forced destruction is used.
</description>
*)
METHOD Cleanup
IF _CleanupComplete THEN
	RETURN;
END_IF

__TRY

	CASE _Phase OF
		FILE_TEST_DIRECTORY_PHASE.CREATE_DIRECTORY:
			_CleanupComplete := TRUE;
			_CleanupSucceeded := TRUE;
			_Phase := FILE_TEST_DIRECTORY_PHASE.COMPLETE;

		FILE_TEST_DIRECTORY_PHASE.WAIT_FOR_DIRECTORY:
			_Phase := FILE_TEST_DIRECTORY_PHASE.DRAIN_CREATION;

		FILE_TEST_DIRECTORY_PHASE.DRAIN_CREATION:

			IF _CreateDirectory.State.Running THEN
				_CreateDirectory.Cancel();
				_CreateDirectory.Execute();
			END_IF

			IF NOT _CreateDirectory.State.Running THEN

				IF _CreateDirectory.State.Stopped AND_THEN _CreateDirectory.FinalStopReason.WorkDone THEN
					_OwnsDirectory := TRUE;
					_Phase := FILE_TEST_DIRECTORY_PHASE.READY;
				ELSE
					_CleanupMessage := 'Interrupted creation has unknown effects; inspect the unowned directory';
					_CleanupComplete := TRUE;
					_Phase := FILE_TEST_DIRECTORY_PHASE.COMPLETE;
				END_IF

			END_IF

		FILE_TEST_DIRECTORY_PHASE.READY:
			_Phase := FILE_TEST_DIRECTORY_PHASE.DELETE_FIRST_FILE;

		FILE_TEST_DIRECTORY_PHASE.DELETE_FIRST_FILE:

			IF _FirstFileMayExist THEN

				IF _DeleteFirstFile.State.Ready THEN
					_DeleteFirstFile.FilePath := FirstFilePath;
					_DeleteFirstFile.PathType := Tc2_System.E_OpenPath.PATH_GENERIC;
					_DeleteFirstFile.Timeout := T#2S;

					IF NOT _DeleteFirstFile.Start() THEN
						_CleanupMessage := 'Artifact deletion: Start refused; inspect the scenario directory';
						_Phase := FILE_TEST_DIRECTORY_PHASE.DELETE_SECOND_FILE;
						RETURN;
					END_IF

				END_IF

				_DeleteFirstFile.Execute();

				IF NOT _DeleteFirstFile.State.Stopped THEN
					RETURN;
				END_IF

				IF NOT _DeleteFirstFile.FinalStopReason.WorkDone THEN
					_CleanupMessage := TO_STRING(_DeleteFirstFile.FinalStopReason.Message);
				END_IF

			END_IF

			_Phase := FILE_TEST_DIRECTORY_PHASE.DELETE_SECOND_FILE;

		FILE_TEST_DIRECTORY_PHASE.DELETE_SECOND_FILE:

			IF _SecondFileMayExist THEN

				IF _DeleteSecondFile.State.Ready THEN
					_DeleteSecondFile.FilePath := SecondFilePath;
					_DeleteSecondFile.PathType := Tc2_System.E_OpenPath.PATH_GENERIC;
					_DeleteSecondFile.Timeout := T#2S;

					IF NOT _DeleteSecondFile.Start() THEN
						_CleanupMessage := 'Artifact deletion: Start refused; inspect the scenario directory';
						_Phase := FILE_TEST_DIRECTORY_PHASE.REMOVE_DIRECTORY;
						RETURN;
					END_IF

				END_IF

				_DeleteSecondFile.Execute();

				IF NOT _DeleteSecondFile.State.Stopped THEN
					RETURN;
				END_IF

				IF NOT _DeleteSecondFile.FinalStopReason.WorkDone THEN
					_CleanupMessage := TO_STRING(_DeleteSecondFile.FinalStopReason.Message);
				END_IF

			END_IF

			_Phase := FILE_TEST_DIRECTORY_PHASE.REMOVE_DIRECTORY;

		FILE_TEST_DIRECTORY_PHASE.REMOVE_DIRECTORY:

			IF _RemoveDirectory.State.Ready THEN
				_RemoveDirectory.DirectoryPath := _DirectoryPath;
				_RemoveDirectory.PathType := Tc2_System.E_OpenPath.PATH_GENERIC;
				_RemoveDirectory.Timeout := T#2S;

				IF NOT _RemoveDirectory.Start() THEN
					_CleanupMessage := 'Directory cleanup: Start refused';
					_CleanupComplete := TRUE;
					_Phase := FILE_TEST_DIRECTORY_PHASE.COMPLETE;
					RETURN;
				END_IF

			END_IF

			_RemoveDirectory.Execute();

			IF _RemoveDirectory.State.Stopped THEN
				_CleanupSucceeded := _RemoveDirectory.FinalStopReason.WorkDone;

				IF _CleanupSucceeded THEN
					_OwnsDirectory := FALSE;
				ELSE
					_CleanupMessage := TO_STRING(_RemoveDirectory.FinalStopReason.Message);
				END_IF

				_CleanupComplete := TRUE;
				_Phase := FILE_TEST_DIRECTORY_PHASE.COMPLETE;
			END_IF

	END_CASE

__CATCH
	(* Persistent tasks remain available; a later call resumes the interrupted cleanup phase. *)
	_CleanupMessage := 'Exception interrupted scenario cleanup; keep cycling and inspect the directory';
__ENDTRY
END_METHOD

(*!
<summary>Rearms this fixture after successful cleanup without performing directory I/O.</summary>
<description>
Call from the owning task after cleanup completed successfully and all scenario managers are idle.
Returns TRUE for a fresh fixture. Returns FALSE if cleanup is pending, ownership is unresolved, or a
native task refuses reset. On partial task reset the fixture keeps its completed state and diagnostics.
</description>
*)
METHOD Reset : BOOL
IF _Phase = FILE_TEST_DIRECTORY_PHASE.CREATE_DIRECTORY THEN
	Reset := TRUE;
	RETURN;
END_IF

IF NOT _CleanupComplete OR_ELSE NOT _CleanupSucceeded OR_ELSE _OwnsDirectory THEN
	RETURN;
END_IF

IF NOT _CreateDirectory.Reset()
	OR_ELSE NOT _DeleteFirstFile.Reset()
	OR_ELSE NOT _DeleteSecondFile.Reset()
	OR_ELSE NOT _RemoveDirectory.Reset()
THEN
	RETURN;
END_IF

_PreparationFailed := FALSE;
_PreparationMessage := TOF_Core.Strings.Empty;
_CleanupComplete := FALSE;
_CleanupSucceeded := FALSE;
_CleanupMessage := TOF_Core.Strings.Empty;
_FirstFileMayExist := FALSE;
_SecondFileMayExist := FALSE;
_Phase := FILE_TEST_DIRECTORY_PHASE.CREATE_DIRECTORY;
Reset := TRUE;
END_METHOD

(*!
<summary>Reports exclusive ownership after successful ordinary creation.</summary>
*)
PROPERTY Prepared : BOOL
GET
Prepared := _Phase = FILE_TEST_DIRECTORY_PHASE.READY AND_THEN _OwnsDirectory;
END_GET
END_PROPERTY

(*!
<summary>Reports refusal, native failure or an exception during preparation.</summary>
*)
PROPERTY PreparationFailed : BOOL
GET
PreparationFailed := _PreparationFailed;
END_GET
END_PROPERTY

(*!
<summary>Copies the retained preparation diagnostic.</summary>
*)
PROPERTY PreparationMessage : STRING(255)
GET
PreparationMessage := _PreparationMessage;
END_GET
END_PROPERTY

(*!
<summary>Reports that cleanup attempts ended, including unsuccessful attempts.</summary>
*)
PROPERTY CleanupComplete : BOOL
GET
CleanupComplete := _CleanupComplete;
END_GET
END_PROPERTY

(*!
<summary>Reports directory removal or cleanup before any creation request.</summary>
*)
PROPERTY CleanupSucceeded : BOOL
GET
CleanupSucceeded := _CleanupSucceeded;
END_GET
END_PROPERTY

(*!
<summary>Copies any retained cleanup error; inspect it together with DirectoryPath.</summary>
*)
PROPERTY CleanupMessage : STRING(255)
GET
CleanupMessage := _CleanupMessage;
END_GET
END_PROPERTY

(*!
<summary>Copies the fixed scenario directory path.</summary>
*)
PROPERTY DirectoryPath : STRING(255)
GET
DirectoryPath := _DirectoryPath;
END_GET
END_PROPERTY

(*!
<summary>Copies the first fixed artifact path inside this scenario directory.</summary>
*)
PROPERTY FirstFilePath : STRING(255)
GET
FirstFilePath := TOF_Core.Strings.Concat255(_DirectoryPath, '\First.txt');
END_GET
END_PROPERTY

(*!
<summary>Copies the second fixed artifact path inside this scenario directory.</summary>
*)
PROPERTY SecondFilePath : STRING(255)
GET
SecondFilePath := TOF_Core.Strings.Concat255(_DirectoryPath, '\Second.txt');
END_GET
END_PROPERTY

(*!
<summary>Stops cleanup attempts for the first artifact after confirmed removal.</summary>
<description>
The caller has successfully deleted or renamed this artifact while retaining exclusive directory ownership.
This notification performs no filesystem check and must not be used for an uncertain or cancelled operation.
</description>
*)
METHOD ConfirmFirstFileAbsent
_FirstFileMayExist := FALSE;
END_METHOD

(*!
<summary>Stops cleanup attempts for the second artifact after confirmed removal.</summary>
<description>
The caller has successfully deleted or renamed this artifact while retaining exclusive directory ownership.
This notification performs no filesystem check and must not be used for an uncertain or cancelled operation.
</description>
*)
METHOD ConfirmSecondFileAbsent
_SecondFileMayExist := FALSE;
END_METHOD

END_FUNCTION_BLOCK

// ---- Tests/Files/FileTestRoot.TcPOU
(*
SPDX-FileCopyrightText: © 2026 Oleksandr Tiutyk <trofimich@gmail.com>
SPDX-License-Identifier: MIT
License: https://opensource.org/license/mit
*)

(*!
<summary>Prepares the shared filesystem test root for both test runners.</summary>
<description>
The test controller calls Execute once per cycle from its owner task before the test runners. All filesystem suites
borrow the resulting readiness; they must not create the root independently. The root is reserved for tests
and is never removed. A deadline reports failure and subsequent calls continue cancelling and draining the
pending native task. Prepared does not certify physical resource release after a native abort error.
</description>
*)

{attribute 'no_explicit_call' := 'Use Execute from the test controller'}
PROGRAM FileTestRoot
VAR CONSTANT
	//! <summary>Root reserved for independently owned filesystem scenario directories.</summary>
	_RootPath : STRING(255) := 'C:\OpenFrameworkTests';
END_VAR
VAR
	_CreateRoot : TOF_FileSystem.CreateDirectoryIfNotExists(name := "prepareFileTestRoot");
	_Started : BOOL;
	_Prepared : BOOL;
	_FailureMessage : STRING(255);
	_Deadline : Tc2_Standard.TON;
END_VAR

(*!
<summary>Advances root preparation or its failure cleanup without abandoning pending I/O.</summary>
*)
METHOD Execute
IF _Prepared THEN
	RETURN;
END_IF

__TRY

	IF _FailureMessage <> TOF_Core.Strings.Empty THEN

		IF _CreateRoot.State.Running THEN
			_CreateRoot.Cancel();
			_CreateRoot.Execute();
		END_IF

		RETURN;
	END_IF

	_Deadline(IN := TRUE, PT := T#10S);

	IF NOT _Started THEN
		_CreateRoot.DirectoryPath := _RootPath;
		_CreateRoot.PathType := Tc2_System.E_OpenPath.PATH_GENERIC;
		_CreateRoot.Timeout := T#2S;

		IF NOT _CreateRoot.Start() THEN
			_FailureMessage := 'Filesystem test root: Start refused';
			RETURN;
		END_IF

		_Started := TRUE;
	END_IF

	_CreateRoot.Execute();

	IF _CreateRoot.State.Stopped THEN

		IF _CreateRoot.FinalStopReason.WorkDone THEN
			_Prepared := TRUE;
		ELSE
			_FailureMessage := TOF_Core.Strings.Concat255(
				'Filesystem test root: ',
				TO_STRING(_CreateRoot.FinalStopReason.Message)
			);
		END_IF

	ELSIF _Deadline.Q THEN
		_FailureMessage := 'Filesystem test root preparation exceeded 10 seconds';
		_CreateRoot.Cancel();
	END_IF

__CATCH
	(* Record failure without diagnostic callbacks; later cycles still drain the persistent task. *)
	_FailureMessage := 'Exception interrupted filesystem test root preparation';
__ENDTRY
END_METHOD

(*!
<summary>Reports successful completion of shared root preparation.</summary>
*)
PROPERTY Prepared : BOOL
GET
Prepared := _Prepared;
END_GET
END_PROPERTY

(*!
<summary>Copies the retained preparation failure; empty while pending or successful.</summary>
*)
PROPERTY FailureMessage : STRING(255)
GET
FailureMessage := _FailureMessage;
END_GET
END_PROPERTY

(*!
<summary>Reports pending root preparation or stopping that still requires cyclic Execute.</summary>
*)
PROPERTY Running : BOOL
GET
Running := _CreateRoot.State.Running;
END_GET
END_PROPERTY

END_PROGRAM

// ---- Tests/Files/LexicalPathValidationTest.TcPOU
(*
SPDX-FileCopyrightText: © 2026 Oleksandr Tiutyk <trofimich@gmail.com>
SPDX-License-Identifier: MIT
License: https://opensource.org/license/mit
*)

(*!
<summary>Checks lexical path acceptance, rejection diagnostics and full-length path handling.</summary>
<description>Uses fixed expectations and requires no filesystem I/O or shared test directory.</description>
*)

{attribute 'no_explicit_call' := 'do not call this function block directly'}
FUNCTION_BLOCK LexicalPathValidationTest EXTENDS TOF_Testing.SingleCycleTest
VAR CONSTANT
	//! <summary>Lexical inputs and their independent expected directory and file results.</summary>
	_PathCases : ARRAY [0..23] OF PATH_VALIDATION_TEST_CASE := [
		(Path := '', DirectoryAccepted := FALSE, FileAccepted := FALSE),
		(Path := 'C:\file.txt', DirectoryAccepted := TRUE, FileAccepted := TRUE),
		(Path := 'C:\', DirectoryAccepted := TRUE, FileAccepted := FALSE),
		(Path := '/', DirectoryAccepted := TRUE, FileAccepted := FALSE),
		(Path := '\', DirectoryAccepted := TRUE, FileAccepted := FALSE),
		(Path := 'file/', DirectoryAccepted := TRUE, FileAccepted := FALSE),
		(Path := 'file\', DirectoryAccepted := TRUE, FileAccepted := FALSE),
		(Path := '\\server\share\file', DirectoryAccepted := TRUE, FileAccepted := TRUE),
		(Path := '//server/share/file', DirectoryAccepted := TRUE, FileAccepted := TRUE),
		(Path := 'a//b', DirectoryAccepted := FALSE, FileAccepted := FALSE),
		(Path := 'C:relative', DirectoryAccepted := FALSE, FileAccepted := FALSE),
		(Path := '1:\file', DirectoryAccepted := FALSE, FileAccepted := FALSE),
		(Path := 'file^name', DirectoryAccepted := FALSE, FileAccepted := FALSE),
		(Path := '.', DirectoryAccepted := TRUE, FileAccepted := TRUE),
		(Path := '..', DirectoryAccepted := TRUE, FileAccepted := TRUE),
		(Path := 'CON', DirectoryAccepted := TRUE, FileAccepted := TRUE),
		(Path := 'file ', DirectoryAccepted := TRUE, FileAccepted := TRUE),
		(Path := 'file.', DirectoryAccepted := TRUE, FileAccepted := TRUE),
		(Path := 'file?x', DirectoryAccepted := FALSE, FileAccepted := FALSE),
		(Path := 'file$01', DirectoryAccepted := FALSE, FileAccepted := FALSE),
		(Path := 'C:/file', DirectoryAccepted := TRUE, FileAccepted := TRUE),
		(Path := '\\', DirectoryAccepted := TRUE, FileAccepted := FALSE),
		(Path := 'a\\b', DirectoryAccepted := FALSE, FileAccepted := FALSE),
		(Path := 'C:\123|456', DirectoryAccepted := FALSE, FileAccepted := FALSE)
	];
END_VAR
VAR_STAT
	{attribute 'hide'}
	_ClassName : STRING := __POUNAME();
END_VAR

(*!
<summary>Borrows the concrete class name for the lifetime of this instance.</summary>
*)
{attribute 'monitoring' := 'call'}
PROPERTY ClassName : REFERENCE TO STRING
GET
ClassName REF= _ClassName;
END_GET
END_PROPERTY

(*!
<summary>Runs the path matrix and the full-length separator checks in a single cycle.</summary>
*)
METHOD PROTECTED ExecuteTest
checkPathMatrix();
checkFullLengthPath();
END_METHOD

(*!
<summary>Checks both lexical outcomes and requires a fresh diagnostic on every rejection.</summary>
<description>Reads fixed cases from the test fixture. Reserved names and dot components are checked only against the lexical filter.</description>
*)
METHOD PRIVATE checkPathMatrix
VAR
	accepted : BOOL;
	errorMessage : WSTRING(255);
	pathForDiagnostic : WSTRING(255);
	i : DINT;
END_VAR
FOR i := LOWER_BOUND(_PathCases, 1) TO UPPER_BOUND(_PathCases, 1) DO
	pathForDiagnostic := TO_WSTRING(_PathCases[i].Path);
	errorMessage := TOF_Core.WideStrings.Empty;
	accepted := TOF_FileSystem.PathHelper.IsValidDirectoryPath(
		directoryPath := _PathCases[i].Path,
		errorMessage => errorMessage
	);
	Assert.ThatBool(
		actual := accepted,
		message := TOF_Core.WideStrings.ConcatFit255("Directory path: [", pathForDiagnostic, "]")
	).ToBe(expected := _PathCases[i].DirectoryAccepted);

	IF NOT _PathCases[i].DirectoryAccepted THEN
		Assert.ThatWideString(
			actual := errorMessage,
			message := TOF_Core.WideStrings.ConcatFit255("Missing directory rejection diagnostic: [", pathForDiagnostic, "]")
		).NotToBe(expected := TOF_Core.WideStrings.Empty);
	END_IF

	errorMessage := TOF_Core.WideStrings.Empty;
	accepted := TOF_FileSystem.PathHelper.IsValidFilePath(filePath := _PathCases[i].Path, errorMessage => errorMessage);
	Assert.ThatBool(
		actual := accepted,
		message := TOF_Core.WideStrings.ConcatFit255("File path: [", pathForDiagnostic, "]")
	).ToBe(expected := _PathCases[i].FileAccepted);

	IF NOT _PathCases[i].FileAccepted THEN
		Assert.ThatWideString(
			actual := errorMessage,
			message := TOF_Core.WideStrings.ConcatFit255("Missing file rejection diagnostic: [", pathForDiagnostic, "]")
		).NotToBe(expected := TOF_Core.WideStrings.Empty);
	END_IF
END_FOR
END_METHOD

(*!
<summary>Checks the last payload byte of a full-length path for the file and directory rules.</summary>
*)
METHOD PRIVATE checkFullLengthPath
VAR
	path : Tc2_System.T_MaxString;
	lastPayloadIndex : UDINT;
	i : UDINT;
END_VAR
// The final byte of the IEC string is reserved for its terminator.
lastPayloadIndex := SIZEOF(path) - 2;

// SA0175: The boundary fixture is a byte string containing ASCII characters.
{analysis -175}
FOR i := 0 TO lastPayloadIndex DO
	path[i] := Tc2_System.F_ToASC(str := 'a');
END_FOR

path[lastPayloadIndex + 1] := 0;
{analysis +175}

Assert.ThatBool(
	actual := TOF_FileSystem.PathHelper.IsValidFilePath(filePath := path),
	message := "A 255-byte lexical filename must pass"
).IsTrue();

{analysis -175}
path[lastPayloadIndex] := Tc2_System.F_ToASC(str := '/');
{analysis +175}

Assert.ThatBool(
	actual := TOF_FileSystem.PathHelper.IsValidFilePath(filePath := path),
	message := "A separator at the last payload byte must be rejected for a file"
).IsFalse();
Assert.ThatBool(
	actual := TOF_FileSystem.PathHelper.IsValidDirectoryPath(directoryPath := path),
	message := "A trailing directory separator is permitted lexically"
).IsTrue();
END_METHOD

(*!
<summary>Borrows the compiler-initialized namespace for the lifetime of this instance.</summary>
*)
{attribute 'monitoring' := 'call'}
PROPERTY NamespaceName : REFERENCE TO STRING
GET
NamespaceName REF= CurrentNamespace.Name;
END_GET
END_PROPERTY

(*!
<summary>Reports the complete concrete instance size in bytes.</summary>
*)
{attribute 'monitoring' := 'call'}
PROPERTY SelfSize : ULINT
GET
SelfSize := XSIZEOF(THIS^);
END_GET
END_PROPERTY

END_FUNCTION_BLOCK

// ---- Tests/Files/FileSystemContractTest.TcPOU
(*
SPDX-FileCopyrightText: © 2026 Oleksandr Tiutyk <trofimich@gmail.com>
SPDX-License-Identifier: MIT
License: https://opensource.org/license/mit
*)

(*!
<summary>Groups the deterministic filesystem contract scenarios.</summary>
<description>
Owns six persistent child tests and their fixed parent associations. Use in one task without reentry.
Do not copy the group or modify its borrowed Children array. The cases require no shared test directory.
</description>
*)

{attribute 'no_assign'}
{attribute 'no_explicit_call' := 'do not call this function block directly'}
FUNCTION_BLOCK FileSystemContractTest EXTENDS TOF_Testing.TestGroup<6>
VAR_STAT
	{attribute 'hide'}
	_ClassName : STRING := __POUNAME();
END_VAR
VAR
	_DefaultNamesAndReuse : FileSystemDefaultNamesTest(name := "DefaultNamesAndReuse", parent := THIS^);
	_UnboundContentFailures : FileSystemUnboundContentTest(name := "UnboundContentFailures", parent := THIS^);
	_LoadBufferPreconditions : FileSystemLoadBufferTest(name := "LoadBufferPreconditions", parent := THIS^);
	_QueueBindingRules : FileSystemQueueBindingTest(name := "QueueBindingRules", parent := THIS^);
	_ExceptionClonePayloads : FileSystemExceptionCloneTest(name := "ExceptionClonePayloads", parent := THIS^);
	_ManagerStartRefusal : FileSystemManagerStartRefusalTest(name := "ManagerStartRefusal", parent := THIS^);

	_Children : ARRAY [0.._ChildCount - 1] OF TOF_Testing.ITestElement :=
	[
		_DefaultNamesAndReuse,
		_UnboundContentFailures,
		_LoadBufferPreconditions,
		_QueueBindingRules,
		_ExceptionClonePayloads,
		_ManagerStartRefusal
	];
END_VAR

//! <summary>Borrows the fixed array of this concrete group; do not modify it.</summary>
{attribute 'monitoring' := 'call'}
PROPERTY Children : REFERENCE TO ARRAY [0.._ChildCount - 1] OF TOF_Testing.ITestElement
GET
Children REF= _Children;
END_GET
END_PROPERTY

//! <summary>Borrows the concrete class name for the lifetime of this instance; callers must not modify it.</summary>
{attribute 'monitoring' := 'call'}
PROPERTY ClassName : REFERENCE TO STRING
GET
ClassName REF= _ClassName;
END_GET
END_PROPERTY

//! <summary>Borrows the compiler-initialized namespace; callers must not modify the returned reference.</summary>
{attribute 'monitoring' := 'call'}
PROPERTY NamespaceName : REFERENCE TO STRING
GET
NamespaceName REF= CurrentNamespace.Name;
END_GET
END_PROPERTY

//! <summary>Reports the complete concrete instance size, excluding separately allocated storage.</summary>
{attribute 'monitoring' := 'call'}
PROPERTY SelfSize : ULINT
GET
SelfSize := XSIZEOF(THIS^);
END_GET
END_PROPERTY

END_FUNCTION_BLOCK

// ---- Tests/Files/FileSystemDefaultNamesTest.TcPOU
(*
SPDX-FileCopyrightText: © 2026 Oleksandr Tiutyk <trofimich@gmail.com>
SPDX-License-Identifier: MIT
License: https://opensource.org/license/mit
*)

(*!
<summary>Checks all sixteen default names and cancellation/reset stability without starting native I/O.</summary>
<description>
The fixture belongs to the runner task and is kept between runs. The test drives no native file requests.
</description>
*)

{attribute 'no_assign'}
{attribute 'no_explicit_call' := 'do not call this function block directly'}
FUNCTION_BLOCK FileSystemDefaultNamesTest EXTENDS TOF_Testing.SingleCycleTest
VAR_STAT
	{attribute 'hide'}
	_ClassName : STRING := __POUNAME();
END_VAR
VAR
	_CheckDirectory : TOF_FileSystem.CheckDirectoryExists(name := "");
	_CreateDirectory : TOF_FileSystem.CreateDirectory(name := "");
	_CreateIfAbsent : TOF_FileSystem.CreateDirectoryIfNotExists(name := "");
	_RemoveDirectory : TOF_FileSystem.RemoveEmptyDirectory(name := "");
	_RemoveIfPresent : TOF_FileSystem.RemoveEmptyDirectoryIfExists(name := "");
	_DeleteFile : TOF_FileSystem.DeleteFile(name := "");
	_RenameFile : TOF_FileSystem.RenameFile(name := "");
	_LoadFile : TOF_FileSystem.LoadFile(name := "");
	_Manager : TOF_FileSystem.FileContentManager(name := "");
	_CheckEof : TOF_FileSystem.CheckEndOfFile(name := "");
	_GetPosition : TOF_FileSystem.GetPositionInFile(name := "");
	_SetPosition : TOF_FileSystem.SetPositionInFile(name := "");
	_ReadBytes : TOF_FileSystem.ReadBytesFromFile(name := "");
	_ReadString : TOF_FileSystem.ReadString255FromFile(name := "");
	_WriteBytes : TOF_FileSystem.WriteBytesToFile(name := "");
	_WriteString : TOF_FileSystem.WriteString255ToFile(name := "");
	_ExplicitDirectory : TOF_FileSystem.CreateDirectory(name := "Explicit directory");
	_ExplicitManager : TOF_FileSystem.FileContentManager(name := "Explicit manager");
	_ExplicitRead : TOF_FileSystem.ReadBytesFromFile(name := "Explicit read");

	_Tasks : ARRAY [0..15] OF TOF_Tasks.ITask :=
	[
		_CheckDirectory,
		_CreateDirectory,
		_CreateIfAbsent,
		_RemoveDirectory,
		_RemoveIfPresent,
		_DeleteFile,
		_RenameFile,
		_LoadFile,
		_Manager,
		_CheckEof,
		_GetPosition,
		_SetPosition,
		_ReadBytes,
		_ReadString,
		_WriteBytes,
		_WriteString
	];
END_VAR

